REGION Network 6: Mode
   // 0NA,1Manual, 2Auto, 3Step, 4OneCycle, 5Runn, 6Error
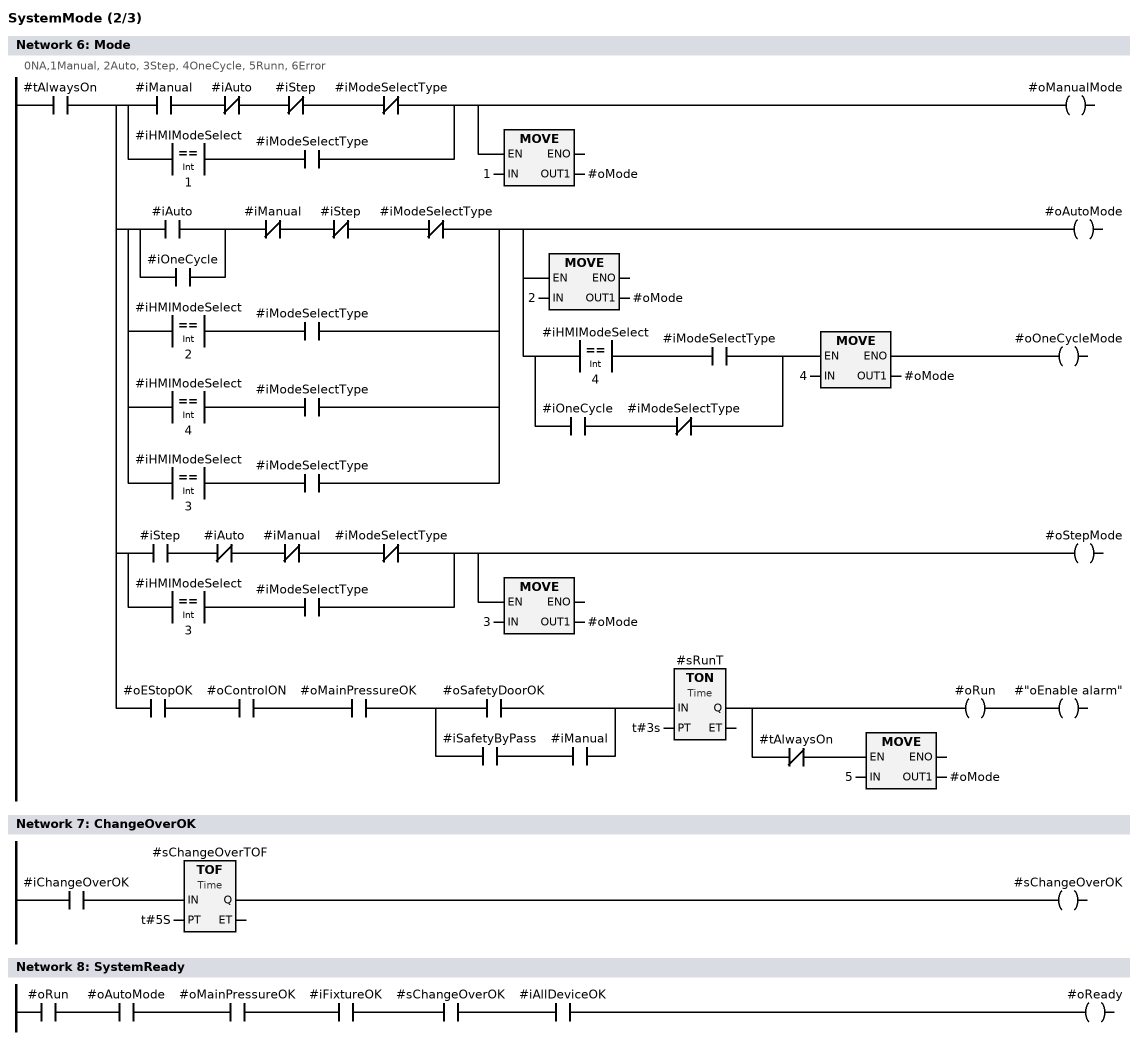
   RUNG wire#powerrail
      Contact( #tAlwaysOn )
      wire#w1
      Contact( #iManual )
      I_Contact( #iAuto )
      I_Contact( #iStep )
      I_Contact( #iModeSelectType )
      wire#w2
      Coil( #oManualMode )
   END_RUNG
   RUNG wire#w1
      { S7_Templates := "SrcType := Int" } EQ_Contact(in1 := #iHMIModeSelect, in2 := 1)
      Contact( #iModeSelectType )
   END_RUNG wire#w2
   RUNG wire#w2
      { S7_GenerateENO := "TRUE" } Move(in := 1, out1 => #oMode)
   END_RUNG
   RUNG wire#w1
      Contact( #iAuto )
      wire#w3
      I_Contact( #iManual )
      I_Contact( #iStep )
      I_Contact( #iModeSelectType )
      wire#w4
      Coil( #oAutoMode )
   END_RUNG
   RUNG wire#w1
      Contact( #iOneCycle )
   END_RUNG wire#w3
   RUNG wire#w1
      { S7_Templates := "SrcType := Int" } EQ_Contact(in1 := #iHMIModeSelect, in2 := 2)
      Contact( #iModeSelectType )
   END_RUNG wire#w4
   RUNG wire#w1
      { S7_Templates := "SrcType := Int" } EQ_Contact(in1 := #iHMIModeSelect, in2 := 4)
      Contact( #iModeSelectType )
   END_RUNG wire#w4
   RUNG wire#w1
      { S7_Templates := "SrcType := Int" } EQ_Contact(in1 := #iHMIModeSelect, in2 := 3)
      Contact( #iModeSelectType )
   END_RUNG wire#w4
   RUNG wire#w4
      { S7_GenerateENO := "TRUE" } Move(in := 2, out1 => #oMode)
   END_RUNG
   RUNG wire#w4
      { S7_Templates := "SrcType := Int" } EQ_Contact(in1 := #iHMIModeSelect, in2 := 4)
      Contact( #iModeSelectType )
      wire#w5
      { S7_GenerateENO := "TRUE" } Move(in := 4, out1 => #oMode)
      Coil( #oOneCycleMode )
   END_RUNG
   RUNG wire#w4
      Contact( #iOneCycle )
      I_Contact( #iModeSelectType )
   END_RUNG wire#w5
   RUNG wire#w1
      Contact( #iStep )
      I_Contact( #iAuto )
      I_Contact( #iManual )
      I_Contact( #iModeSelectType )
      wire#w6
      Coil( #oStepMode )
   END_RUNG
   RUNG wire#w1
      { S7_Templates := "SrcType := Int" } EQ_Contact(in1 := #iHMIModeSelect, in2 := 3)
      Contact( #iModeSelectType )
   END_RUNG wire#w6
   RUNG wire#w6
      { S7_GenerateENO := "TRUE" } Move(in := 3, out1 => #oMode)
   END_RUNG
   RUNG wire#w1
      Contact( #oEStopOK )
      Contact( #oControlON )
      Contact( #oMainPressureOK )
      wire#w7
      Contact( #oSafetyDoorOK )
      wire#w8
      { S7_Templates := "time_type := Time" } #sRunT.TON(pt := t#3s, et =>)
      wire#w9
      Coil( #oRun )
      Coil( #"oEnable alarm" )
   END_RUNG
   RUNG wire#w7
      Contact( #iSafetyByPass )
      Contact( #iManual )
   END_RUNG wire#w8
   RUNG wire#w9
      I_Contact( #tAlwaysOn )
      { S7_GenerateENO := "TRUE" } Move(in := 5, out1 => #oMode)
   END_RUNG
   // the same network as SCL:
   // ENO of a box is taken as its EN; it also drops when the box reports an error
   #oManualMode := #tAlwaysOn AND ((#iManual AND NOT #iAuto AND NOT #iStep AND NOT #iModeSelectType) OR ((#iHMIModeSelect = 1) AND #iModeSelectType));
   IF #oManualMode THEN #oMode := 1; END_IF;
   #oAutoMode := #tAlwaysOn AND (((#iAuto OR #iOneCycle) AND NOT #iManual AND NOT #iStep AND NOT #iModeSelectType) OR ((#iHMIModeSelect = 2) AND #iModeSelectType) OR ((#iHMIModeSelect = 4) AND #iModeSelectType) OR ((#iHMIModeSelect = 3) AND #iModeSelectType));
   IF #oAutoMode THEN #oMode := 2; END_IF;
   #_w1 := #oAutoMode AND (((#iHMIModeSelect = 4) AND #iModeSelectType) OR (#iOneCycle AND NOT #iModeSelectType));
   IF #_w1 THEN #oMode := 4; END_IF;
   #oOneCycleMode := #_w1;
   #oStepMode := #tAlwaysOn AND ((#iStep AND NOT #iAuto AND NOT #iManual AND NOT #iModeSelectType) OR ((#iHMIModeSelect = 3) AND #iModeSelectType));
   IF #oStepMode THEN #oMode := 3; END_IF;
   #sRunT(IN := #tAlwaysOn AND #oEStopOK AND #oControlON AND #oMainPressureOK AND (#oSafetyDoorOK OR (#iSafetyByPass AND #iManual)),   // TON
          PT := t#3s);
   #oRun := #sRunT.Q;
   #"oEnable alarm" := #sRunT.Q;
   IF #sRunT.Q AND NOT #tAlwaysOn THEN #oMode := 5; END_IF;
END_REGION

REGION Network 7: ChangeOverOK
   RUNG wire#powerrail
      Contact( #iChangeOverOK )
      { S7_Templates := "time_type := Time" } #sChangeOverTOF.TOF(pt := t#5S, et =>)
      Coil( #sChangeOverOK )
   END_RUNG
   // the same network as SCL:
   #sChangeOverTOF(IN := #iChangeOverOK, PT := t#5S);   // TOF
   #sChangeOverOK := #sChangeOverTOF.Q;
END_REGION

REGION Network 8: SystemReady
   RUNG wire#powerrail
      Contact( #oRun )
      Contact( #oAutoMode )
      Contact( #oMainPressureOK )
      Contact( #iFixtureOK )
      Contact( #sChangeOverOK )
      Contact( #iAllDeviceOK )
      Coil( #oReady )
   END_RUNG
   // the same network as SCL:
   #oReady := #oRun AND #oAutoMode AND #oMainPressureOK AND #iFixtureOK AND #sChangeOverOK AND #iAllDeviceOK;
END_REGION

REGION Network 9: SystemStatus
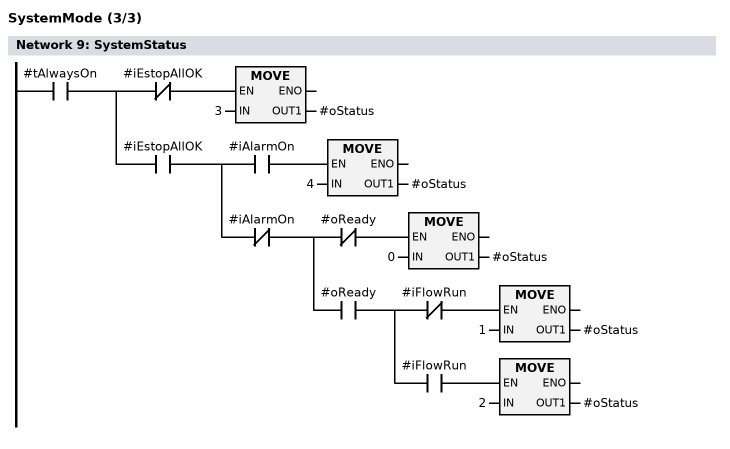
   RUNG wire#powerrail
      Contact( #tAlwaysOn )
      wire#w1
      I_Contact( #iEstopAllOK )
      Move(in := 3, out1 => #oStatus)
   END_RUNG
   RUNG wire#w1
      Contact( #iEstopAllOK )
      wire#w2
      Contact( #iAlarmOn )
      Move(in := 4, out1 => #oStatus)
   END_RUNG
   RUNG wire#w2
      I_Contact( #iAlarmOn )
      wire#w3
      I_Contact( #oReady )
      Move(in := 0, out1 => #oStatus)
   END_RUNG
   RUNG wire#w3
      Contact( #oReady )
      wire#w4
      I_Contact( #iFlowRun )
      Move(in := 1, out1 => #oStatus)
   END_RUNG
   RUNG wire#w4
      Contact( #iFlowRun )
      Move(in := 2, out1 => #oStatus)
   END_RUNG
   // the same network as SCL:
   IF #tAlwaysOn AND NOT #iEstopAllOK THEN #oStatus := 3; END_IF;
   #_w1 := #tAlwaysOn AND #iEstopAllOK;
   IF #_w1 AND #iAlarmOn THEN #oStatus := 4; END_IF;
   #_w2 := #_w1 AND NOT #iAlarmOn;
   IF #_w2 AND NOT #oReady THEN #oStatus := 0; END_IF;
   #_w3 := #_w2 AND #oReady;
   IF #_w3 AND NOT #iFlowRun THEN #oStatus := 1; END_IF;
   IF #_w3 AND #iFlowRun THEN #oStatus := 2; END_IF;
END_REGION
END_FUNCTION_BLOCK

FUNCTION_BLOCK "AutoProcessDataPopUp"   // FB1666, SCL
{ S7_Optimized_Access := 'TRUE' }
// stored: AutoNumber false, MemoryReserve 100, SetENOAutomatically false
   VAR_IN_OUT
      idx { ExternalAccessible := 'False'; ExternalVisible := 'False'; ExternalWritable := 'False'} : Int;
   END_VAR
   VAR_TEMP
      DefaultData : "ProcessData";
   END_VAR
BEGIN
   REGION read me
     // ============================================================================
     // PROGRAM START COMMENT
     // ============================================================================
     // EN:
     // FC_AutoProcessPopup handles popup visualization and editing of AutoProcess
     // data based on index from HMI.
     // The function provides:
     //  - automatic data loading from AutoProcessData according to selected index,
     //  - two-step confirmation for safe data overwrite (compare first, write second),
     //  - automatic reset of edit mode when index is changed,
     //  - delete functionality for selected record,
     //  - status bits for HMI to visualize pending changes and confirmation dialogs,
     //  - index range control (1..16).
     //
     // Data flow:
     // AutoProcessData  -> ActualSHowingData  (display mode)
     // ActualSHowingData -> AutoProcessData  (after double confirmation)
     //
     // Usage:
     // Call cyclically 
     // RMS index is taken from AutoProcess_HMI.IndexProcess.
     //
     // ----------------------------------------------------------------------------
     // CZ:
     // FC_AutoProcessPopup obsluhuje zobrazení a editaci dat AutoProcess podle
     // indexu z HMI.
     // Funkce zajišťuje:
     //  - automatické načítání dat z AutoProcessData podle zvoleného indexu,
     //  - dvoukrokové potvrzení zápisu (nejprve porovnání, poté zápis),
     //  - automatické zrušení editace při změně indexu,
     //  - mazání záznamu podle indexu,
     //  - stavové bity pro HMI (čekající změna, potvrzovací dialog),
     //  - kontrolu rozsahu indexu (1..16).
     //
     // Tok dat:
     // AutoProcessData  -> ActualSHowingData  (zobrazení)
     // ActualSHowingData -> AutoProcessData  (po potvrzení)
     //
     // Použití:
     // Volat cyklicky 
     // Index je čten z AutoProcess_HMI.IndexProcess.
     // ============================================================================

     // Statement section REGION

   END_REGION


   REGION IndexRangeCheck
     // EN: Clamp index to range 1..16
     // CZ: Oříznutí indexu do rozsahu 1..16
     IF #idx < 1 THEN
       #idx := 1;
       "AutoProcess_HMI".IndexProcess := #idx;
     ELSIF #idx > 16 THEN
       #idx := 16;
       "AutoProcess_HMI".IndexProcess := #idx;

     END_IF;
   END_REGION


   REGION IndexHandling
     // ---------------------------------------------------------------------------
     // EN: Detect index change and reset edit session
     // CZ: Detekce změny indexu a zrušení editace
     // ---------------------------------------------------------------------------
     #idx := "AutoProcess_HMI".IndexProcess;

     IF #idx <> "AutoProcess_HMI".Data_handling.LastIndex THEN
       "AutoProcess_HMI".Data_handling.UpdateData_switch := FALSE;
       "AutoProcess_HMI".Data_handling.UpdateData_Confirm := FALSE;
       "AutoProcess_HMI".Data_handling.FinalConfirm_Write := FALSE;
       "AutoProcess_HMI".Data_handling.ConfirmDialogActive := FALSE;
       "AutoProcess_HMI".Data_handling.ChangePending := FALSE;
       "AutoProcess_HMI".Data_handling.DeleteData := FALSE;
       "AutoProcess_HMI".Data_handling.LastIndex := #idx;
     END_IF;
   END_REGION



   REGION ShowData
     // ---------------------------------------------------------------------------
     // EN: Copy data to HMI if edit mode is inactive
     // CZ: Zobrazování dat – pokud není editace, kopíruj data z DB
     // ---------------------------------------------------------------------------
     IF NOT "AutoProcess_HMI".Data_handling.UpdateData_switch THEN
       CASE #idx OF
         1:
           "AutoProcess_HMI".ActualSHowingData := "AutoProcessData".A_ScanRotate;
         2:
           "AutoProcess_HMI".ActualSHowingData := "AutoProcessData".F_Robot1Grip1;
         3:
           "AutoProcess_HMI".ActualSHowingData := "AutoProcessData".F_Robot1Grip2;
         4:
           "AutoProcess_HMI".ActualSHowingData := "AutoProcessData".B_Press1;
         5:
           "AutoProcess_HMI".ActualSHowingData := "AutoProcessData".C_Glue;
         6:
           "AutoProcess_HMI".ActualSHowingData := "AutoProcessData".F_Robot2Grip1;
         7:
           "AutoProcess_HMI".ActualSHowingData := "AutoProcessData".F_Robot2Grip2;
         8:
           "AutoProcess_HMI".ActualSHowingData := "AutoProcessData".C_GlueNGBuffer;
         9:
           "AutoProcess_HMI".ActualSHowingData := "AutoProcessData".C_MagnScanNGBuffer;
         10:
           "AutoProcess_HMI".ActualSHowingData := "AutoProcessData".B_Press2;
         11:
           "AutoProcess_HMI".ActualSHowingData := "AutoProcessData".F_Robot3Grip1;
         12:
           "AutoProcess_HMI".ActualSHowingData := "AutoProcessData".F_Robot3Grip2;
         13:
           "AutoProcess_HMI".ActualSHowingData := "AutoProcessData".H_ShafeLine;
         14:
           "AutoProcess_HMI".ActualSHowingData := "AutoProcessData".J_ShafeLine;
         15:
           "AutoProcess_HMI".ActualSHowingData := "AutoProcessData".K_ShafeLine;
         16:
           "AutoProcess_HMI".ActualSHowingData := "AutoProcessData".L_ShafeLine;
         ELSE
           ;
           // EN: invalid index / CZ: neplatný index
       END_CASE;
     END_IF;
   END_REGION



   REGION FirstConfirm
     // ---------------------------------------------------------------------------
     // EN: First confirmation → enable compare dialog
     // CZ: První potvrzení → aktivace porovnávacího dialogu
     // ---------------------------------------------------------------------------
     IF "AutoProcess_HMI".Data_handling.UpdateData_switch
       AND "AutoProcess_HMI".Data_handling.UpdateData_Confirm
       AND NOT "AutoProcess_HMI".Data_handling.ConfirmDialogActive THEN

       "AutoProcess_HMI".Data_handling.ConfirmDialogActive := TRUE;
       "AutoProcess_HMI".Data_handling.ChangePending := TRUE;

       "AutoProcess_HMI".Data_handling.UpdateData_Confirm := FALSE;
     END_IF;
   END_REGION



   REGION FinalWrite
     // ---------------------------------------------------------------------------
     // EN: Final confirmation → write to data DB
     // CZ: Finální potvrzení → zápis do DB
     // ---------------------------------------------------------------------------
     IF "AutoProcess_HMI".Data_handling.ConfirmDialogActive
       AND "AutoProcess_HMI".Data_handling.FinalConfirm_Write THEN

       CASE #idx OF
         1:
           "AutoProcessData".A_ScanRotate := "AutoProcess_HMI".ActualSHowingData;
         2:
           "AutoProcessData".F_Robot1Grip1 := "AutoProcess_HMI".ActualSHowingData;
         3:
           "AutoProcessData".F_Robot1Grip2 := "AutoProcess_HMI".ActualSHowingData;
         4:
           "AutoProcessData".B_Press1 := "AutoProcess_HMI".ActualSHowingData;
         5:
           "AutoProcessData".C_Glue := "AutoProcess_HMI".ActualSHowingData;
         6:
           "AutoProcessData".F_Robot2Grip1 := "AutoProcess_HMI".ActualSHowingData;
         7:
           "AutoProcessData".F_Robot2Grip2 := "AutoProcess_HMI".ActualSHowingData;
         8:
           "AutoProcessData".C_GlueNGBuffer := "AutoProcess_HMI".ActualSHowingData;
         9:
           "AutoProcessData".C_MagnScanNGBuffer := "AutoProcess_HMI".ActualSHowingData;
         10:
           "AutoProcessData".B_Press2 := "AutoProcess_HMI".ActualSHowingData;
         11:
           "AutoProcessData".F_Robot3Grip1 := "AutoProcess_HMI".ActualSHowingData;
         12:
           "AutoProcessData".F_Robot3Grip2 := "AutoProcess_HMI".ActualSHowingData;
         13:
           "AutoProcessData".H_ShafeLine := "AutoProcess_HMI".ActualSHowingData;
         14:
           "AutoProcessData".J_ShafeLine := "AutoProcess_HMI".ActualSHowingData;
         15:
           "AutoProcessData".K_ShafeLine := "AutoProcess_HMI".ActualSHowingData;
         16:
           "AutoProcessData".L_ShafeLine := "AutoProcess_HMI".ActualSHowingData;
         ELSE
           ;
       END_CASE;

       // reset flags after write
       "AutoProcess_HMI".Data_handling.ConfirmDialogActive := FALSE;
       "AutoProcess_HMI".Data_handling.ChangePending := FALSE;
       "AutoProcess_HMI".Data_handling.FinalConfirm_Write := FALSE;
       "AutoProcess_HMI".Data_handling.UpdateData_switch := FALSE;
     END_IF;
   END_REGION



   REGION DeleteData
     // ---------------------------------------------------------------------------
     // EN: Delete selected Record (reset to default struct)
     // CZ: Smazání záznamu – vynulování struktury
     // ---------------------------------------------------------------------------
     IF "AutoProcess_HMI".Data_handling.DeleteData AND
       "AutoProcess_HMI".Data_handling.FinalConfirm_Write
       THEN

       CASE #idx OF
         1:
           "AutoProcessData".A_ScanRotate := #DefaultData;
         2:
           "AutoProcessData".F_Robot1Grip1 := #DefaultData;
         3:
           "AutoProcessData".F_Robot1Grip2 := #DefaultData;
         4:
           "AutoProcessData".B_Press1 := #DefaultData;
         5:
           "AutoProcessData".C_Glue := #DefaultData;
         6:
           "AutoProcessData".F_Robot2Grip1 := #DefaultData;
         7:
           "AutoProcessData".F_Robot2Grip2 := #DefaultData;
         8:
           "AutoProcessData".C_GlueNGBuffer := #DefaultData;
         9:
           "AutoProcessData".C_MagnScanNGBuffer := #DefaultData;
         10:
           "AutoProcessData".B_Press2 := #DefaultData;
         11:
           "AutoProcessData".F_Robot3Grip1 := #DefaultData;
         12:
           "AutoProcessData".F_Robot3Grip2 := #DefaultData;
         13:
           "AutoProcessData".H_ShafeLine := #DefaultData;
         14:
           "AutoProcessData".J_ShafeLine := #DefaultData;
         15:
           "AutoProcessData".K_ShafeLine := #DefaultData;
         16:
           "AutoProcessData".L_ShafeLine := #DefaultData;
         ELSE
           ;
       END_CASE;

       // reset delete + editing states
       "AutoProcess_HMI".Data_handling.DeleteData := FALSE;
       "AutoProcess_HMI".Data_handling.UpdateData_switch := FALSE;
       "AutoProcess_HMI".Data_handling.UpdateData_Confirm := FALSE;
       "AutoProcess_HMI".Data_handling.FinalConfirm_Write := FALSE;
       "AutoProcess_HMI".Data_handling.ConfirmDialogActive := FALSE;
       "AutoProcess_HMI".Data_handling.ChangePending := FALSE;
     END_IF;
   END_REGION

   REGION StationProductIcons
     // EN: Set icon bits if station contains product (PartStatus <> 0)
     // CZ: Nastavení bitů ikony – stanice má kus, pokud PartStatus <> 0

     // 1 – A_ScanRotate
     "AutoProcess_HMI".StationHasProduct[1] :=
     "AutoProcessData".A_ScanRotate.PartStatus <> 0;

     // 2 – F_Robot1Grip1
     "AutoProcess_HMI".StationHasProduct[2] :=
     "AutoProcessData".F_Robot1Grip1.PartStatus <> 0;

     // 3 – F_Robot1Grip2
     "AutoProcess_HMI".StationHasProduct[3] :=
     "AutoProcessData".F_Robot1Grip2.PartStatus <> 0;

     // 4 – B_Press1
     "AutoProcess_HMI".StationHasProduct[4] :=
     "AutoProcessData".B_Press1.PartStatus <> 0;

     // 5 – C_Glue
     "AutoProcess_HMI".StationHasProduct[5] :=
     "AutoProcessData".C_Glue.PartStatus <> 0;

     // 6 – F_Robot2Grip1
     "AutoProcess_HMI".StationHasProduct[6] :=
     "AutoProcessData".F_Robot2Grip1.PartStatus <> 0;

     // 7 – F_Robot2Grip2
     "AutoProcess_HMI".StationHasProduct[7] :=
     "AutoProcessData".F_Robot2Grip2.PartStatus <> 0;

     // 8 – C_GlueNGBuffer
     "AutoProcess_HMI".StationHasProduct[8] :=
     "AutoProcessData".C_GlueNGBuffer.PartStatus <> 0;

     // 9 – C_MagnScanNGBuffer
     "AutoProcess_HMI".StationHasProduct[9] :=
     "AutoProcessData".C_MagnScanNGBuffer.PartStatus <> 0;

     // 10 – B_Press2
     "AutoProcess_HMI".StationHasProduct[10] :=
     "AutoProcessData".B_Press2.PartStatus <> 0;

     // 11 – F_Robot3Grip1
     "AutoProcess_HMI".StationHasProduct[11] :=
     "AutoProcessData".F_Robot3Grip1.PartStatus <> 0;

     // 12 – F_Robot3Grip2
     "AutoProcess_HMI".StationHasProduct[12] :=
     "AutoProcessData".F_Robot3Grip2.PartStatus <> 0;

     // 13 – H_ShafeLine
     "AutoProcess_HMI".StationHasProduct[13] :=
     "AutoProcessData".H_ShafeLine.PartStatus <> 0;

     // 14 – J_ShafeLine
     "AutoProcess_HMI".StationHasProduct[14] :=
     "AutoProcessData".J_ShafeLine.PartStatus <> 0;

     // 15 – K_ShafeLine
     "AutoProcess_HMI".StationHasProduct[15] :=
     "AutoProcessData".K_ShafeLine.PartStatus <> 0;

     // 16 – L_ShafeLine
     "AutoProcess_HMI".StationHasProduct[16] :=
     "AutoProcessData".L_ShafeLine.PartStatus <> 0;

   END_REGION
END_FUNCTION_BLOCK

ORGANIZATION_BLOCK "02_Warm Restart"   // OB100, LAD, Startup
TITLE = "Complete Restart"
{ S7_Optimized_Access := 'FALSE' }
AUTHOR : RCS
// 1.该部分用户可以根据系统的需要将CPU第一次扫描需要执行的逻辑写在此处
// stored: AutoNumber false, SetENOAutomatically false
   VAR_TEMP
      OB100_EV_CLASS : Byte;   // 16#13, Event class 1, Entering event state, Event logged in diagnostic buffer
      OB100_STRTUP : Byte;   // 16#81/82/83/84 Method of startup
      OB100_PRIORITY : Byte;   // Priority of OB Execution
      OB100_OB_NUMBR : Byte;   // 100 (Organization block 100, OB100)
      OB100_RESERVED_1 : Byte;   // Reserved for system
      OB100_RESERVED_2 : Byte;   // Reserved for system
      OB100_STOP : Word;   // Event that caused CPU to stop (16#4xxx)
      OB100_STRT_INFO : DWord;   // Information on how system started
      OB100_DATE_TIME : Date_And_Time;   // Date and time OB100 started
   END_VAR
BEGIN

REGION Network 1
   // 系统程序段无需改动
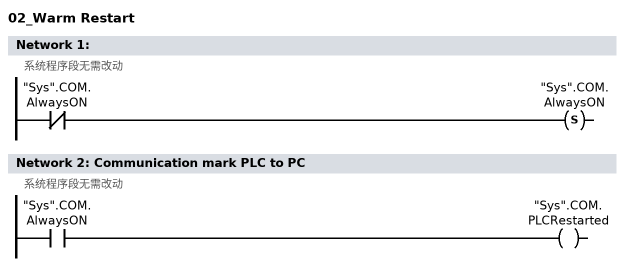
   RUNG wire#powerrail
      I_Contact( "Sys".COM.AlwaysON )
      S_Coil( "Sys".COM.AlwaysON )
   END_RUNG
   // the same network as SCL:
   IF NOT "Sys".COM.AlwaysON THEN "Sys".COM.AlwaysON := TRUE; END_IF;
END_REGION

REGION Network 2: Communication mark PLC to PC
   // 系统程序段无需改动
   RUNG wire#powerrail
      Contact( "Sys".COM.AlwaysON )
      Coil( "Sys".COM.PLCRestarted )
   END_RUNG
   // the same network as SCL:
   "Sys".COM.PLCRestarted := "Sys".COM.AlwaysON;
END_REGION

NETWORK
TITLE = 

      L     1;
      T     "Station_Sys".Status.ModeSV;

END_ORGANIZATION_BLOCK

ORGANIZATION_BLOCK "03_CYC_INT2"   // OB32, LAD, CyclicInterrupt
TITLE = "Cyclic Interrupt"
{ S7_Optimized_Access := 'FALSE' }
// stored: AutoNumber false, SetENOAutomatically false
   VAR_TEMP
      OB32_EV_CLASS : Byte;   // Bits 0-3 = 1 (Coming event), Bits 4-7 = 1 (Event class 1)
      OB32_STRT_INF : Byte;   // 16#33 (OB 32 has started)
      OB32_PRIORITY : Byte;   // Priority of OB Execution
      OB32_OB_NUMBR : Byte;   // 32 (Organization block 32, OB32)
      OB32_RESERVED_1 : Byte;   // Reserved for system
      OB32_RESERVED_2 : Byte;   // Reserved for system
      OB32_PHS_OFFSET : Int;   // Phase offset (integer, milliseconds)
      OB32_RESERVED_3 : Int;   // Reserved for system
      OB32_EXC_FREQ : Int;   // Frequency of execution (msec)
      OB32_DATE_TIME : Date_And_Time;   // Date and time OB32 started
   END_VAR
BEGIN

REGION Network 1
   // //Keep resource code
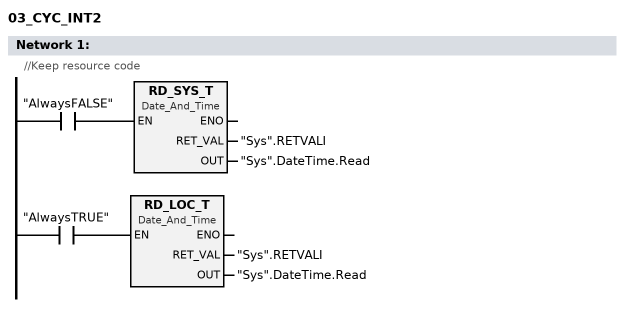
   RUNG wire#powerrail
      Contact( "AlwaysFALSE" )
      { S7_Templates := "date_type := Date_And_Time" } RD_SYS_T(RET_VAL => "Sys".RETVALI, OUT => "Sys".DateTime.Read)
   END_RUNG
   RUNG wire#powerrail
      Contact( "AlwaysTRUE" )
      { S7_Templates := "date_type := Date_And_Time" } RD_LOC_T(RET_VAL => "Sys".RETVALI, OUT => "Sys".DateTime.Read)
   END_RUNG
   // the same network as SCL:
   IF "AlwaysFALSE" THEN "Sys".RETVALI := RD_SYS_T(OUT => "Sys".DateTime.Read); END_IF;
   IF "AlwaysTRUE" THEN "Sys".RETVALI := RD_LOC_T(OUT => "Sys".DateTime.Read); END_IF;
END_REGION

NETWORK
TITLE = Diagnostic
//      CALL  "Diagnostic"
//         iCPUType :=2
//         iDBNum   :=3001
//         iOffset  :=0


END_ORGANIZATION_BLOCK

ORGANIZATION_BLOCK "04_CYC_INT5"   // OB35, LAD, CyclicInterrupt
TITLE = "Cyclic Interrupt"
{ S7_Optimized_Access := 'FALSE' }
// stored: AutoNumber false, SetENOAutomatically false
   VAR_TEMP
      OB35_EV_CLASS : Byte;   // Bits 0-3 = 1 (Coming event), Bits 4-7 = 1 (Event class 1)
      OB35_STRT_INF : Byte;   // 16#36 (OB 35 has started)
      OB35_PRIORITY : Byte;   // Priority of OB Execution
      OB35_OB_NUMBR : Byte;   // 35 (Organization block 35, OB35)
      OB35_RESERVED_1 : Byte;   // Reserved for system
      OB35_RESERVED_2 : Byte;   // Reserved for system
      OB35_PHASE_OFFSET : Word;   // Phase offset (msec)
      OB35_RESERVED_3 : Int;   // Reserved for system
      OB35_EXC_FREQ : Int;   // Frequency of execution (msec)
      OB35_DATE_TIME : Date_And_Time;   // Date and time OB35 started
   END_VAR
BEGIN
END_ORGANIZATION_BLOCK

ORGANIZATION_BLOCK "05_MOD_ERR"   // OB122, STL, IOAccessError
TITLE = "Module Access Error"
{ S7_Optimized_Access := 'FALSE' }
   VAR_TEMP
      OB122_EV_CLASS : Byte;   // 16#29, Event class 2, Entering event state, Internal fault event
      OB122_SW_FLT : Byte;   // 16#XX Software error code
      OB122_PRIORITY : Byte;   // Priority of OB Execution
      OB122_OB_NUMBR : Byte;   // 122 (Organization block 122, OB122)
      OB122_BLK_TYPE : Byte;   // 16#88/8C/8E Type of block fault occured in
      OB122_MEM_AREA : Byte;   // Memory area where access error occured
      OB122_MEM_ADDR : Word;   // Memory address where access error occured
      OB122_BLK_NUM : Word;   // Block number in which error occured
      OB122_PRG_ADDR : Word;   // Program address where error occured
      OB122_DATE_TIME : Date_And_Time;   // Date and time OB1 started
   END_VAR
BEGIN
END_ORGANIZATION_BLOCK

ORGANIZATION_BLOCK "07_CYCL_FLT"   // OB80, STL, TimeErrorInterrupt
TITLE = "Cycle Time Fault"
{ S7_Optimized_Access := 'FALSE' }
   VAR_TEMP
      OB80_EV_CLASS : Byte;   // 16#35, Event class 3, Entering event state, Internal fault event
      OB80_FLT_ID : Byte;   // 16#XX, Fault identifcation code
      OB80_PRIORITY : Byte;   // Priority of OB Execution
      OB80_OB_NUMBR : Byte;   // 80 (Organization block 80, OB80)
      OB80_RESERVED_1 : Byte;   // Reserved for system
      OB80_RESERVED_2 : Byte;   // Reserved for system
      OB80_ERROR_INFO : Word;   // Error information on event
      OB80_ERR_EV_CLASS : Byte;   // Class of event causing error
      OB80_ERR_EV_NUM : Byte;   // Number of event causing error
      OB80_OB_PRIORITY : Byte;   // Priority of OB causing error
      OB80_OB_NUM : Byte;   // Number of OB causing error
      OB80_DATE_TIME : Date_And_Time;   // Date and time OB80 started
   END_VAR
BEGIN
END_ORGANIZATION_BLOCK

ORGANIZATION_BLOCK "08_HW_INT0"   // OB40, LAD, HardwareInterrupt
TITLE = "Hardware Interrupt"
{ S7_Optimized_Access := 'FALSE' }
// stored: AutoNumber false, SetENOAutomatically false
   VAR_TEMP
      OB40_EV_CLASS : Byte;   // Bits 0-3 = 1 (Coming event), Bits 4-7 = 1 (Event class 1)
      OB40_STRT_INF : Byte;   // 16#41 (OB 40 has started)
      OB40_PRIORITY : Byte;   // Priority of OB Execution
      OB40_OB_NUMBR : Byte;   // 40 (Organization block 40, OB40)
      OB40_RESERVED_1 : Byte;   // Reserved for system
      OB40_IO_FLAG : Byte;   // 16#54 (input module), 16#55 (output module)
      OB40_MDL_ADDR : Word;   // Base address of module initiating interrupt
      OB40_POINT_ADDR : DWord;   // Interrupt status of the module
      OB40_DATE_TIME : Date_And_Time;   // Date and time OB40 started
   END_VAR
BEGIN
END_ORGANIZATION_BLOCK

ORGANIZATION_BLOCK "09_I/O_FLT1"   // OB82, STL, DiagnosticErrorInterrupt
TITLE = "I/O Point Fault"
{ S7_Optimized_Access := 'FALSE' }
   VAR_TEMP
      OB82_EV_CLASS : Byte;   // 16#39, Event class 3, Entering event state, Internal fault event
      OB82_FLT_ID : Byte;   // 16#XX, Fault identifcation code
      OB82_PRIORITY : Byte;   // Priority of OB Execution
      OB82_OB_NUMBR : Byte;   // 82 (Organization block 82, OB82)
      OB82_RESERVED_1 : Byte;   // Reserved for system
      OB82_IO_FLAG : Byte;   // Input (01010100), Output (01010101)
      OB82_MDL_ADDR : Int;   // Base address of module with fault
      OB82_MDL_DEFECT : Bool;   // Module defective
      OB82_INT_FAULT : Bool;   // Internal fault
      OB82_EXT_FAULT : Bool;   // External fault
      OB82_PNT_INFO : Bool;   // Point information
      OB82_EXT_VOLTAGE : Bool;   // External voltage low
      OB82_FLD_CONNCTR : Bool;   // Field wiring connector missing
      OB82_NO_CONFIG : Bool;   // Module has no configuration data
      OB82_CONFIG_ERR : Bool;   // Module has configuration error
      OB82_MDL_TYPE : Byte;   // Type of module
      OB82_SUB_NDL_ERR : Bool;   // Sub-Module is missing or has error
      OB82_COMM_FAULT : Bool;   // Communication fault
      OB82_MDL_STOP : Bool;   // Module is stopped
      OB82_WTCH_DOG_FLT : Bool;   // Watch dog timer stopped module
      OB82_INT_PS_FLT : Bool;   // Internal power supply fault
      OB82_PRIM_BATT_FLT : Bool;   // Primary battery is in fault
      OB82_BCKUP_BATT_FLT : Bool;   // Backup battery is in fault
      OB82_RESERVED_2 : Bool;   // Reserved for system
      OB82_RACK_FLT : Bool;   // Rack fault, only for bus interface module
      OB82_PROC_FLT : Bool;   // Processor fault
      OB82_EPROM_FLT : Bool;   // EPROM fault
      OB82_RAM_FLT : Bool;   // RAM fault
      OB82_ADU_FLT : Bool;   // ADU fault
      OB82_FUSE_FLT : Bool;   // Fuse fault
      OB82_HW_INTR_FLT : Bool;   // Hardware interupt input in fault
      OB82_RESERVED_3 : Bool;   // Reserved for system
      OB82_DATE_TIME : Date_And_Time;   // Date and time OB82 started
   END_VAR
BEGIN
END_ORGANIZATION_BLOCK

ORGANIZATION_BLOCK "11_PROG_ERR"   // OB121, STL, ProgrammingError
TITLE = "Programming Error"
{ S7_Optimized_Access := 'FALSE' }
   VAR_TEMP
      OB121_EV_CLASS : Byte;   // 16#25, Event class 2, Entering event state, Internal fault event
      OB121_SW_FLT : Byte;   // 16#XX Software programming fault
      OB121_PRIORITY : Byte;   // Priority of OB Execution
      OB121_OB_NUMBR : Byte;   // 121 (Organization block 121, OB121)
      OB121_BLK_TYPE : Byte;   // 16#88/8A/8B/8C/8E Type of block fault occured in
      OB121_RESERVED_1 : Byte;   // Reserved for system
      OB121_FLT_REG : Word;   // 16#XX Specific register that caused fault
      OB121_BLK_NUM : Word;   // Number of block that programming fault occured in
      OB121_PRG_ADDR : Word;   // Address in block where programming fault occured
      OB121_DATE_TIME : Date_And_Time;   // Date and time OB121 started
   END_VAR
BEGIN
END_ORGANIZATION_BLOCK

ORGANIZATION_BLOCK "12_RACK_FLT"   // OB86, STL, RackOrStationFailure
TITLE = "Loss Of Rack Fault"
{ S7_Optimized_Access := 'FALSE' }
   VAR_TEMP
      OB86_EV_CLASS : Byte;   // 16#38/39 Event class 3
      OB86_FLT_ID : Byte;   // 16#C1/C4/C5, Fault identifcation code
      OB86_PRIORITY : Byte;   // Priority of OB Execution
      OB86_OB_NUMBR : Byte;   // 86 (Organization block 86, OB86)
      OB86_RESERVED_1 : Byte;   // Reserved for system
      OB86_RESERVED_2 : Byte;   // Reserved for system
      OB86_MDL_ADDR : Word;   // Base address of IM module in rack with fault
      OB86_RACKS_FLTD : Array[0..31] of Bool;
      OB86_DATE_TIME : Date_And_Time;   // Date and time OB86 started
   END_VAR
BEGIN
END_ORGANIZATION_BLOCK

FUNCTION "fcFixtureCheck" : Void   // FC2, LAD
{ S7_Optimized_Access := 'TRUE' }
// stored: SetENOAutomatically false
   VAR_INPUT
      iRecipeSetValue : Byte;   // 配方设定工装值
   END_VAR
   VAR_IN_OUT
      FixtureIDCheck : Struct
         FixtureIDSetValue : Int;
         FixtureIDCheckValue : Int;
         FixtureCheckResult : Bool;
         FixtureCheckUnEnable : Bool;   // 工装检测使能,不需要检测时，给1
      END_STRUCT;
   END_VAR
BEGIN

REGION Network 2: 配方设定工装值 / Formula set tooling values
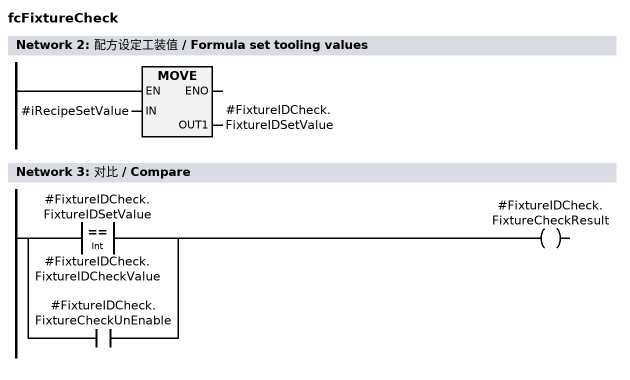
   RUNG wire#powerrail
      Move(in := #iRecipeSetValue, out1 => #FixtureIDCheck.FixtureIDSetValue)
   END_RUNG
   // the same network as SCL:
   #FixtureIDCheck.FixtureIDSetValue := #iRecipeSetValue;
END_REGION

REGION Network 3: 对比 / Compare
   RUNG wire#powerrail
      { S7_Templates := "SrcType := Int" } EQ_Contact(in1 := #FixtureIDCheck.FixtureIDSetValue, in2 := #FixtureIDCheck.FixtureIDCheckValue)
      wire#w1
      Coil( #FixtureIDCheck.FixtureCheckResult )
   END_RUNG
   RUNG wire#powerrail
      Contact( #FixtureIDCheck.FixtureCheckUnEnable )
   END_RUNG wire#w1
   // the same network as SCL:
   #FixtureIDCheck.FixtureCheckResult := (#FixtureIDCheck.FixtureIDSetValue = #FixtureIDCheck.FixtureIDCheckValue) OR #FixtureIDCheck.FixtureCheckUnEnable;
END_REGION
END_FUNCTION

FUNCTION "CylinderModule_V2" : Void   // FC3010, LAD
TITLE = Title
{ S7_Optimized_Access := 'FALSE' }
VERSION : 2.0
// //---------------------------------------------------------------//
// //FunctionName:CylinderV2
// //FunctionDescription:CylinderControl
// //---------------------------------------------------------------//
// //in:
// 
// 	iReset	Bool			reset action
// 	iRun	Bool			system run
// 	iE_stop	Bool			e_stop monitor
// 	iManualMode	Bool		manual mode
// 	iAutoMode	Bool		auto mode
// 	iEnableAlarm	Bool		alarm will popup up
// 	iPulse_100mS	Bool		pulse *100ms
// 	iPulse_1S	Bool		pulse*1s
// 	iCyDBNO	Int	Int		Interface data block number
// 	iCyCounts	Int		total counts of cylinder to be used[must                                                                                                             be>=1 and <=100]
// 
// //inout:
// //out:
// //---------------------------------------------------------------//
// //Version:V2
// //D&T:2016-11-14
// //Group:RCS
// //Author:JM
// //-------------------------Modify1----------------------------------//
// //Version:
// //D&T:2016-11-17
// //Group: RCS
// //Author:
// //Modify:Update cylinder no as output interface
// //-------------------------Modify2----------------------------------//
// //Version:
// //D&T:2022-12-07
// //Group: RCS
// //Author:JM
// //Modify: add action time
// stored: AutoNumber false, SetENOAutomatically false
   VAR_INPUT
      iReset : Bool;   // reset action
      iRun : Bool;   // system run
      iEStop : Bool;   // e_stop monitor
      iManualMode : Bool;   // manual mode
      iAutoMode : Bool;   // auto mode
      iEnableAlarm : Bool;   // alarm will popup up
      iPulse100mS : Bool;   // pulse *100ms
      iPulse1S : Bool;   // pulse*1s
      iError : Bool;   // Outer error force output off
      iGoWorkInterlock : Bool;   // 1=permit motion
      iGoHomeInterlock : Bool;   // 1=permit motion
      iWorkPositionSensor : Bool;   // PLC DI
      iHomePositionSensor : Bool;   // PLC DI
      iValveType : Bool;   // reserve 2022-12-07 / 0 : don`t need holding(2way&3way middle sealing) / 1: need holding(3way middle leaking)
      iManualOutputType : Bool;   // 0 : Output not hold / 1: Output hold (in Manual mode)
      iFaultTime : Int;   // Value*100mS
      iOnPositionTime : Int;   // Value*100mS
   END_VAR
   VAR_OUTPUT
      oGoWP_ButtonActive : Bool;   // For HMI button,indicate can operate go work button
      oGoHP_ButtonActive : Bool;   // For HMI button,indicate can operate go home button
      oCyNo : Byte;
   END_VAR
   VAR_IN_OUT
      ioManualGoWork : Bool;
      ioManualGoHome : Bool;
      ioAutoGoWork : Bool;
      ioAutoGoHome : Bool;
      ioResetOut : Bool;
      ioGoWorkTime : Int;   // Time for going to work position
      ioGoHomeTime : Int;   // time for going to home position
      ioWorkFaultTime : Int;
      ioHomeFaultTime : Int;
      ioBothSensorOnTime : Int;
      ioPulse100mSP : Bool;
      ioAutoGoWorkP : Bool;
      ioAutoGoHomeP : Bool;
      ioGoWork100mSP : Bool;
      ioGoHome100mSP : Bool;
      ioBothSensorOn100mSP : Bool;
      ioAlarm : Bool;
      ioSpare1 : Bool;
      ioSpare2 : Byte;
      ioGoWorkFault : Bool;
      ioGoHomeFault : Bool;
      ioSensorPositionFault : Bool;
      ioGoWorkPosition : Bool;   // PLC DQ
      ioGoHomePosition : Bool;   // PLC DQ
   END_VAR
   VAR_TEMP   // added for the SCL form of the ladder/FBD networks
      _w1 : Bool;
      _w2 : Bool;
      _w3 : Bool;
      _w4 : Bool;
   END_VAR
BEGIN

REGION Network 1: Reset Go Work & Go Home
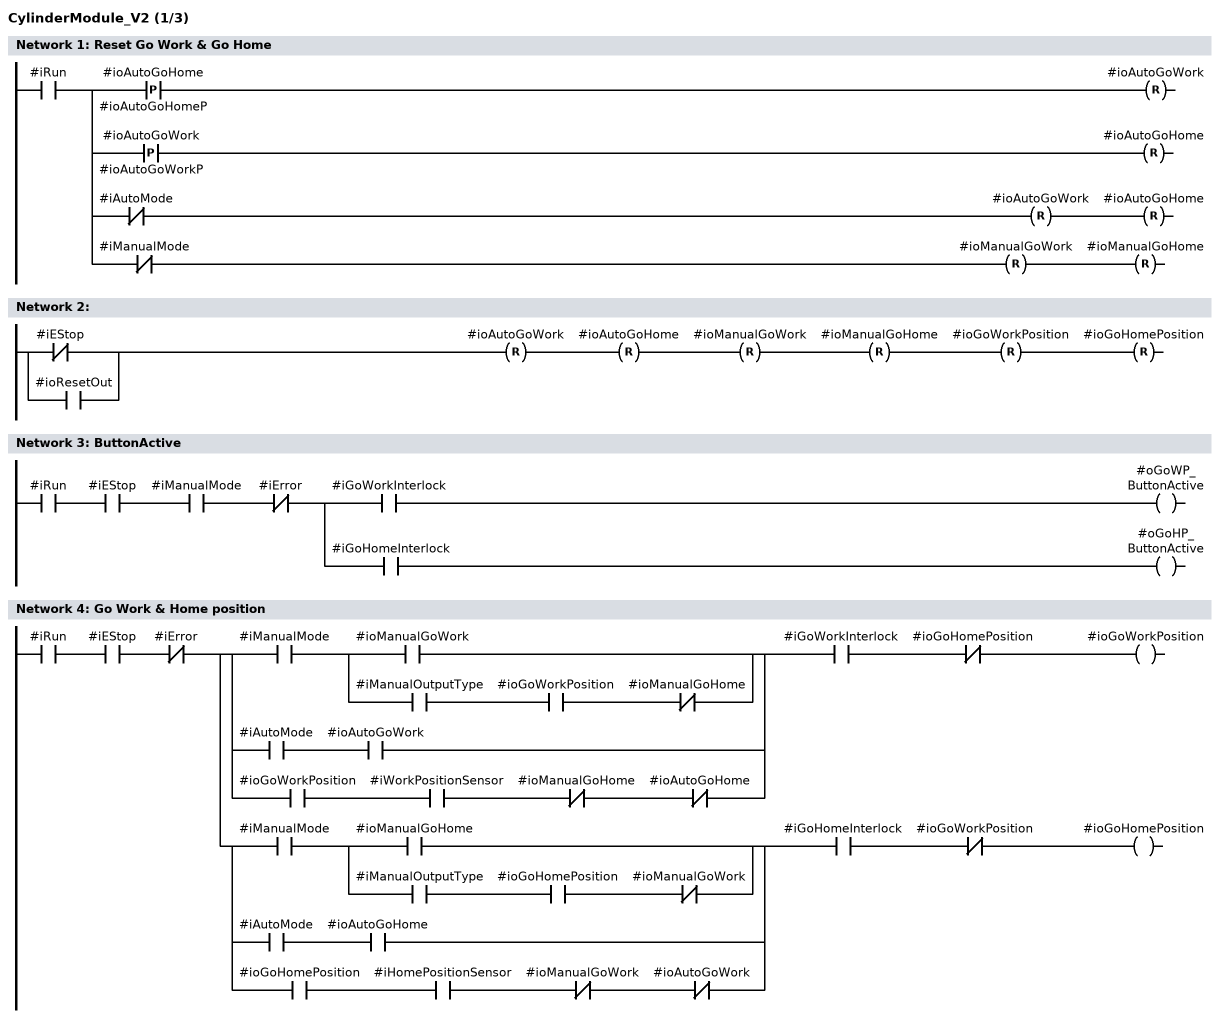
   RUNG wire#powerrail
      Contact( #iRun )
      wire#w1
      P_Contact(operand := #ioAutoGoHome, bit := #ioAutoGoHomeP)
      R_Coil( #ioAutoGoWork )
   END_RUNG
   RUNG wire#w1
      P_Contact(operand := #ioAutoGoWork, bit := #ioAutoGoWorkP)
      R_Coil( #ioAutoGoHome )
   END_RUNG
   RUNG wire#w1
      I_Contact( #iAutoMode )
      R_Coil( #ioAutoGoWork )
      R_Coil( #ioAutoGoHome )
   END_RUNG
   RUNG wire#w1
      I_Contact( #iManualMode )
      R_Coil( #ioManualGoWork )
      R_Coil( #ioManualGoHome )
   END_RUNG
   // the same network as SCL:
   #_w1 := #iRun AND #ioAutoGoHome AND NOT #ioAutoGoHomeP;   // rising edge of #ioAutoGoHome
   #ioAutoGoHomeP := #ioAutoGoHome;
   IF #_w1 THEN #ioAutoGoWork := FALSE; END_IF;
   #_w2 := #iRun AND #ioAutoGoWork AND NOT #ioAutoGoWorkP;   // rising edge of #ioAutoGoWork
   #ioAutoGoWorkP := #ioAutoGoWork;
   IF #_w2 THEN #ioAutoGoHome := FALSE; END_IF;
   IF #iRun AND NOT #iAutoMode THEN
       #ioAutoGoWork := FALSE;
       #ioAutoGoHome := FALSE;
   END_IF;
   IF #iRun AND NOT #iManualMode THEN
       #ioManualGoWork := FALSE;
       #ioManualGoHome := FALSE;
   END_IF;
END_REGION

REGION Network 2
   RUNG wire#powerrail
      I_Contact( #iEStop )
      wire#w1
      R_Coil( #ioAutoGoWork )
      R_Coil( #ioAutoGoHome )
      R_Coil( #ioManualGoWork )
      R_Coil( #ioManualGoHome )
      R_Coil( #ioGoWorkPosition )
      R_Coil( #ioGoHomePosition )
   END_RUNG
   RUNG wire#powerrail
      Contact( #ioResetOut )
   END_RUNG wire#w1
   // the same network as SCL:
   IF NOT #iEStop OR #ioResetOut THEN
       #ioAutoGoWork := FALSE;
       #ioAutoGoHome := FALSE;
       #ioManualGoWork := FALSE;
       #ioManualGoHome := FALSE;
       #ioGoWorkPosition := FALSE;
       #ioGoHomePosition := FALSE;
   END_IF;
END_REGION

REGION Network 3: ButtonActive
   RUNG wire#powerrail
      Contact( #iRun )
      Contact( #iEStop )
      Contact( #iManualMode )
      I_Contact( #iError )
      wire#w1
      Contact( #iGoWorkInterlock )
      Coil( #oGoWP_ButtonActive )
   END_RUNG
   RUNG wire#w1
      Contact( #iGoHomeInterlock )
      Coil( #oGoHP_ButtonActive )
   END_RUNG
   // the same network as SCL:
   #_w1 := #iRun AND #iEStop AND #iManualMode AND NOT #iError;
   #oGoWP_ButtonActive := #_w1 AND #iGoWorkInterlock;
   #oGoHP_ButtonActive := #_w1 AND #iGoHomeInterlock;
END_REGION

REGION Network 4: Go Work & Home position
   RUNG wire#powerrail
      Contact( #iRun )
      Contact( #iEStop )
      I_Contact( #iError )
      wire#w1
      Contact( #iManualMode )
      wire#w2
      Contact( #ioManualGoWork )
      wire#w3
      Contact( #iGoWorkInterlock )
      I_Contact( #ioGoHomePosition )
      Coil( #ioGoWorkPosition )
   END_RUNG
   RUNG wire#w2
      Contact( #iManualOutputType )
      Contact( #ioGoWorkPosition )
      I_Contact( #ioManualGoHome )
   END_RUNG wire#w3
   RUNG wire#w1
      Contact( #iAutoMode )
      Contact( #ioAutoGoWork )
   END_RUNG wire#w3
   RUNG wire#w1
      Contact( #ioGoWorkPosition )
      Contact( #iWorkPositionSensor )
      I_Contact( #ioManualGoHome )
      I_Contact( #ioAutoGoHome )
   END_RUNG wire#w3
   RUNG wire#w1
      Contact( #iManualMode )
      wire#w4
      Contact( #ioManualGoHome )
      wire#w5
      Contact( #iGoHomeInterlock )
      I_Contact( #ioGoWorkPosition )
      Coil( #ioGoHomePosition )
   END_RUNG
   RUNG wire#w4
      Contact( #iManualOutputType )
      Contact( #ioGoHomePosition )
      I_Contact( #ioManualGoWork )
   END_RUNG wire#w5
   RUNG wire#w1
      Contact( #iAutoMode )
      Contact( #ioAutoGoHome )
   END_RUNG wire#w5
   RUNG wire#w1
      Contact( #ioGoHomePosition )
      Contact( #iHomePositionSensor )
      I_Contact( #ioManualGoWork )
      I_Contact( #ioAutoGoWork )
   END_RUNG wire#w5
   // the same network as SCL:
   #_w1 := #iRun AND #iEStop AND NOT #iError;
   #ioGoWorkPosition := #_w1 AND ((#iManualMode AND (#ioManualGoWork OR (#iManualOutputType AND #ioGoWorkPosition AND NOT #ioManualGoHome))) OR (#iAutoMode AND #ioAutoGoWork) OR (#ioGoWorkPosition AND #iWorkPositionSensor AND NOT #ioManualGoHome AND NOT #ioAutoGoHome)) AND #iGoWorkInterlock AND NOT #ioGoHomePosition;
   #ioGoHomePosition := #_w1 AND ((#iManualMode AND (#ioManualGoHome OR (#iManualOutputType AND #ioGoHomePosition AND NOT #ioManualGoWork))) OR (#iAutoMode AND #ioAutoGoHome) OR (#ioGoHomePosition AND #iHomePositionSensor AND NOT #ioManualGoWork AND NOT #ioAutoGoWork)) AND #iGoHomeInterlock AND NOT #ioGoWorkPosition;
END_REGION

REGION Network 5: Go_work_fault
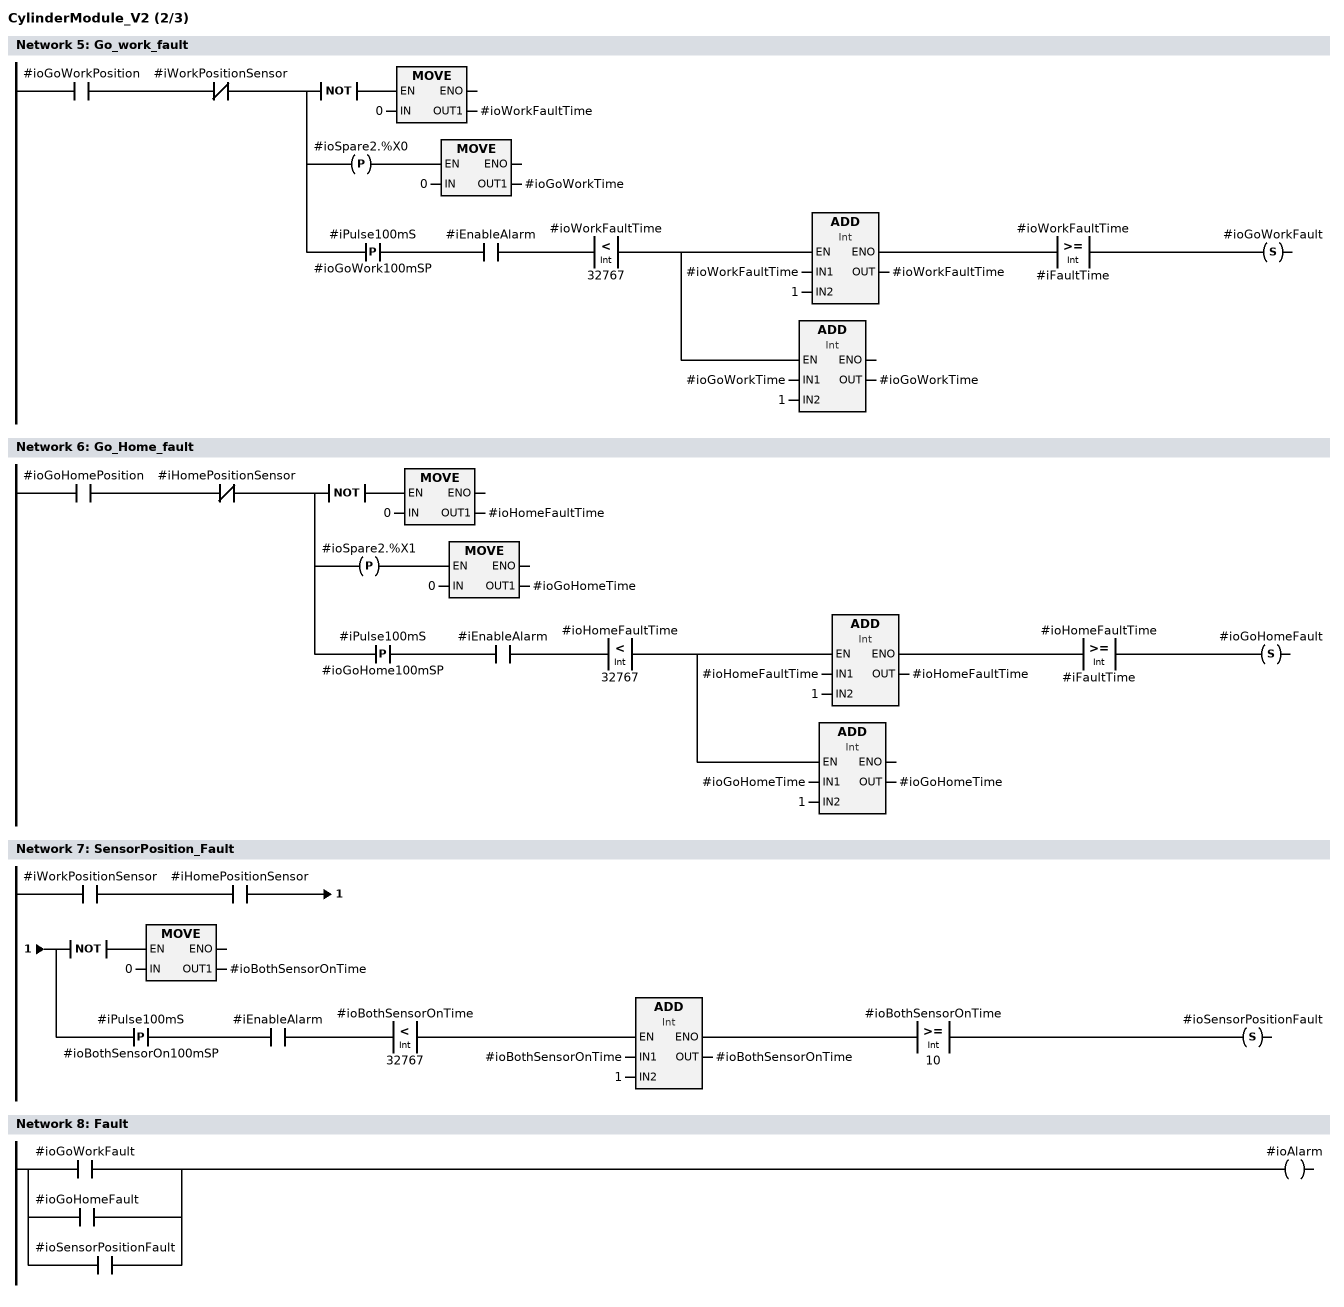
   RUNG wire#powerrail
      Contact( #ioGoWorkPosition )
      I_Contact( #iWorkPositionSensor )
      wire#w1
      Not()
      { S7_GenerateENO := "TRUE" } Move(in := 0, out1 => #ioWorkFaultTime)
   END_RUNG
   RUNG wire#w1
      P_Trig( #ioSpare2.%X0 )
      { S7_GenerateENO := "TRUE" } Move(in := 0, out1 => #ioGoWorkTime)
   END_RUNG
   RUNG wire#w1
      P_Contact(operand := #iPulse100mS, bit := #ioGoWork100mSP)
      Contact( #iEnableAlarm )
      { S7_Templates := "SrcType := Int" } LT_Contact(in1 := #ioWorkFaultTime, in2 := 32767)
      wire#w2
      { S7_Templates := "SrcType := Int"; S7_GenerateENO := "TRUE" } Add(in1 := #ioWorkFaultTime, in2 := 1, out => #ioWorkFaultTime)
      { S7_Templates := "SrcType := Int" } GE_Contact(in1 := #ioWorkFaultTime, in2 := #iFaultTime)
      S_Coil( #ioGoWorkFault )
   END_RUNG
   RUNG wire#w2
      { S7_Templates := "SrcType := Int"; S7_GenerateENO := "TRUE" } Add(in1 := #ioGoWorkTime, in2 := 1, out => #ioGoWorkTime)
   END_RUNG
   // the same network as SCL:
   // ENO of a box is taken as its EN; it also drops when the box reports an error
   #_w1 := #ioGoWorkPosition AND NOT #iWorkPositionSensor;
   IF NOT #_w1 THEN #ioWorkFaultTime := 0; END_IF;
   #_w2 := #_w1 AND NOT #ioSpare2.%X0;   // rising edge
   #ioSpare2.%X0 := #_w1;
   IF #_w2 THEN #ioGoWorkTime := 0; END_IF;
   #_w3 := #_w1 AND #iPulse100mS AND NOT #ioGoWork100mSP;   // rising edge of #iPulse100mS
   #ioGoWork100mSP := #iPulse100mS;
   #_w4 := #_w3 AND #iEnableAlarm AND (#ioWorkFaultTime < 32767);
   IF #_w4 THEN #ioWorkFaultTime := #ioWorkFaultTime + 1; END_IF;
   IF #_w4 AND (#ioWorkFaultTime >= #iFaultTime) THEN #ioGoWorkFault := TRUE; END_IF;
   IF #_w4 THEN #ioGoWorkTime := #ioGoWorkTime + 1; END_IF;
END_REGION

REGION Network 6: Go_Home_fault
   RUNG wire#powerrail
      Contact( #ioGoHomePosition )
      I_Contact( #iHomePositionSensor )
      wire#w1
      Not()
      { S7_GenerateENO := "TRUE" } Move(in := 0, out1 => #ioHomeFaultTime)
   END_RUNG
   RUNG wire#w1
      P_Trig( #ioSpare2.%X1 )
      { S7_GenerateENO := "TRUE" } Move(in := 0, out1 => #ioGoHomeTime)
   END_RUNG
   RUNG wire#w1
      P_Contact(operand := #iPulse100mS, bit := #ioGoHome100mSP)
      Contact( #iEnableAlarm )
      { S7_Templates := "SrcType := Int" } LT_Contact(in1 := #ioHomeFaultTime, in2 := 32767)
      wire#w2
      { S7_Templates := "SrcType := Int"; S7_GenerateENO := "TRUE" } Add(in1 := #ioHomeFaultTime, in2 := 1, out => #ioHomeFaultTime)
      { S7_Templates := "SrcType := Int" } GE_Contact(in1 := #ioHomeFaultTime, in2 := #iFaultTime)
      S_Coil( #ioGoHomeFault )
   END_RUNG
   RUNG wire#w2
      { S7_Templates := "SrcType := Int"; S7_GenerateENO := "TRUE" } Add(in1 := #ioGoHomeTime, in2 := 1, out => #ioGoHomeTime)
   END_RUNG
   // the same network as SCL:
   // ENO of a box is taken as its EN; it also drops when the box reports an error
   #_w1 := #ioGoHomePosition AND NOT #iHomePositionSensor;
   IF NOT #_w1 THEN #ioHomeFaultTime := 0; END_IF;
   #_w2 := #_w1 AND NOT #ioSpare2.%X1;   // rising edge
   #ioSpare2.%X1 := #_w1;
   IF #_w2 THEN #ioGoHomeTime := 0; END_IF;
   #_w3 := #_w1 AND #iPulse100mS AND NOT #ioGoHome100mSP;   // rising edge of #iPulse100mS
   #ioGoHome100mSP := #iPulse100mS;
   #_w4 := #_w3 AND #iEnableAlarm AND (#ioHomeFaultTime < 32767);
   IF #_w4 THEN #ioHomeFaultTime := #ioHomeFaultTime + 1; END_IF;
   IF #_w4 AND (#ioHomeFaultTime >= #iFaultTime) THEN #ioGoHomeFault := TRUE; END_IF;
   IF #_w4 THEN #ioGoHomeTime := #ioGoHomeTime + 1; END_IF;
END_REGION

REGION Network 7: SensorPosition_Fault
   RUNG wire#powerrail
      Contact( #iWorkPositionSensor )
      Contact( #iHomePositionSensor )
      wire#w1
      Not()
      { S7_GenerateENO := "TRUE" } Move(in := 0, out1 => #ioBothSensorOnTime)
   END_RUNG
   RUNG wire#w1
      P_Contact(operand := #iPulse100mS, bit := #ioBothSensorOn100mSP)
      Contact( #iEnableAlarm )
      { S7_Templates := "SrcType := Int" } LT_Contact(in1 := #ioBothSensorOnTime, in2 := 32767)
      { S7_Templates := "SrcType := Int"; S7_GenerateENO := "TRUE" } Add(in1 := #ioBothSensorOnTime, in2 := 1, out => #ioBothSensorOnTime)
      { S7_Templates := "SrcType := Int" } GE_Contact(in1 := #ioBothSensorOnTime, in2 := 10)
      S_Coil( #ioSensorPositionFault )
   END_RUNG
   // the same network as SCL:
   // ENO of a box is taken as its EN; it also drops when the box reports an error
   #_w1 := #iWorkPositionSensor AND #iHomePositionSensor;
   IF NOT #_w1 THEN #ioBothSensorOnTime := 0; END_IF;
   #_w2 := #_w1 AND #iPulse100mS AND NOT #ioBothSensorOn100mSP;   // rising edge of #iPulse100mS
   #ioBothSensorOn100mSP := #iPulse100mS;
   #_w3 := #_w2 AND #iEnableAlarm AND (#ioBothSensorOnTime < 32767);
   IF #_w3 THEN #ioBothSensorOnTime := #ioBothSensorOnTime + 1; END_IF;
   IF #_w3 AND (#ioBothSensorOnTime >= 10) THEN #ioSensorPositionFault := TRUE; END_IF;
END_REGION

REGION Network 8: Fault
   RUNG wire#powerrail
      Contact( #ioGoWorkFault )
      wire#w1
      Coil( #ioAlarm )
   END_RUNG
   RUNG wire#powerrail
      Contact( #ioGoHomeFault )
   END_RUNG wire#w1
   RUNG wire#powerrail
      Contact( #ioSensorPositionFault )
   END_RUNG wire#w1
   // the same network as SCL:
   #ioAlarm := #ioGoWorkFault OR #ioGoHomeFault OR #ioSensorPositionFault;
END_REGION

REGION Network 9: Reset fault
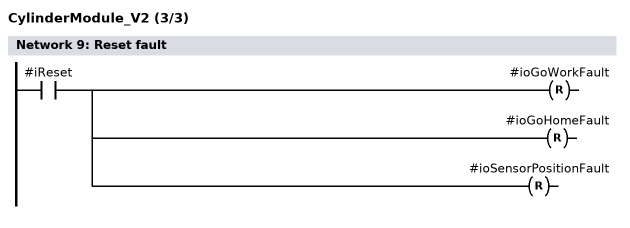
   RUNG wire#powerrail
      Contact( #iReset )
      wire#w1
      R_Coil( #ioGoWorkFault )
   END_RUNG
   RUNG wire#w1
      R_Coil( #ioGoHomeFault )
   END_RUNG
   RUNG wire#w1
      R_Coil( #ioSensorPositionFault )
   END_RUNG
   // the same network as SCL:
   IF #iReset THEN
       #ioGoWorkFault := FALSE;
       #ioGoHomeFault := FALSE;
       #ioSensorPositionFault := FALSE;
   END_IF;
END_REGION
END_FUNCTION

FUNCTION_BLOCK "MaterialGate"   // FB5210, LAD
{ S7_Optimized_Access := 'FALSE' }
// stored: AutoNumber false, SetENOAutomatically false
   VAR_INPUT
      iSysInface : "RCS_SysComInterface_V1";
      "iMaterialGate Opened Monitor" : Bool;   // 安全门打开状态监控
      "iMaterialGate Locked Monitor" : Bool;   // 安全门锁定状态监控
      i1s_Pulse : Bool;   // 1s脉冲信号
      "iMaterialGate AutoLock Timer" : Time := T#1s;   // 安全门自动模式下锁延时
      "iMaterialGate ManualLock Timer" : Time := T#60s;   // 安全门手动模式下锁定延时
   END_VAR
   VAR_OUTPUT
      "oMaterialGate LockedLamp" { ExternalAccessible := 'False'; ExternalVisible := 'False'; ExternalWritable := 'False'} : Bool;   // 安全门解锁输出状态
   END_VAR
   VAR_IN_OUT
      ioMaterialGateLock : Bool;   // 安全门锁定输出
      ioHMI_Interface : "SafetyGateUDT";
   END_VAR
   VAR
      "sMaterialafetyGate Timer" { S7_SetPoint := 'True'} : Array[1..5] of TON_TIME;
      sP_Trig : Array[1..10] of Bool;
      sN_Trig : Array[1..10] of Bool;
      "sMaterialGate UnlockRequest" { ExternalAccessible := 'False'; ExternalVisible := 'False'; ExternalWritable := 'False'} : Bool;   // 安全门开门请求标志位
      "sMaterialGate LockRequest" : Bool;
   END_VAR
   VAR_TEMP
      tAlyways_On : Bool;
      tAlyways_Off : Bool;
   END_VAR
   VAR_TEMP   // added for the SCL form of the ladder/FBD networks
      _w1 : Bool;
      _w2 : Bool;
      _w3 : Bool;
      _w4 : Bool;
      _w5 : Bool;
      _w6 : Bool;
      _w7 : Bool;
   END_VAR
BEGIN

REGION Network 1: #tAlyways_On
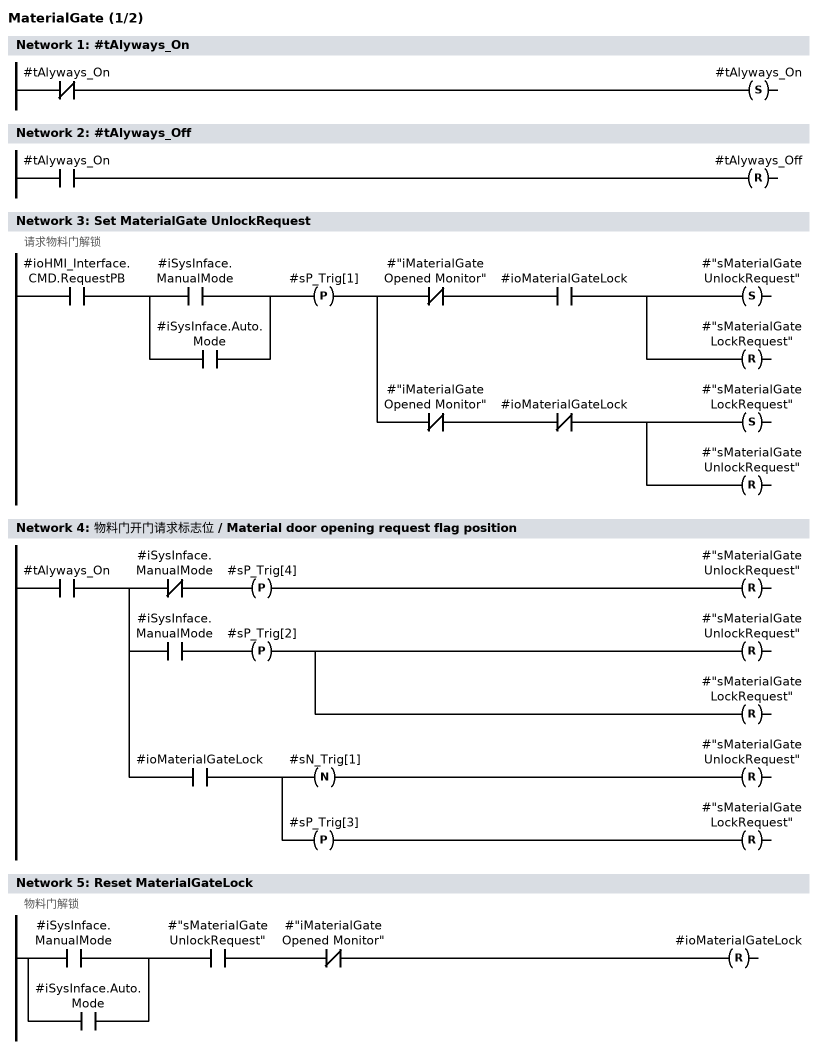
   RUNG wire#powerrail
      I_Contact( #tAlyways_On )
      S_Coil( #tAlyways_On )
   END_RUNG
   // the same network as SCL:
   IF NOT #tAlyways_On THEN #tAlyways_On := TRUE; END_IF;
END_REGION

REGION Network 2: #tAlyways_Off
   RUNG wire#powerrail
      Contact( #tAlyways_On )
      R_Coil( #tAlyways_Off )
   END_RUNG
   // the same network as SCL:
   IF #tAlyways_On THEN #tAlyways_Off := FALSE; END_IF;
END_REGION

REGION Network 3: Set MaterialGate UnlockRequest
   // 请求物料门解锁
   RUNG wire#powerrail
      Contact( #ioHMI_Interface.CMD.RequestPB )
      wire#w1
      Contact( #iSysInface.ManualMode )
      wire#w2
      P_Trig( #sP_Trig[1] )
      wire#w3
      I_Contact( #"iMaterialGate Opened Monitor" )
      Contact( #ioMaterialGateLock )
      wire#w4
      S_Coil( #"sMaterialGate UnlockRequest" )
   END_RUNG
   RUNG wire#w1
      Contact( #iSysInface.Auto.Mode )
   END_RUNG wire#w2
   RUNG wire#w4
      R_Coil( #"sMaterialGate LockRequest" )
   END_RUNG
   RUNG wire#w3
      I_Contact( #"iMaterialGate Opened Monitor" )
      I_Contact( #ioMaterialGateLock )
      wire#w5
      S_Coil( #"sMaterialGate LockRequest" )
   END_RUNG
   RUNG wire#w5
      R_Coil( #"sMaterialGate UnlockRequest" )
   END_RUNG
   // the same network as SCL:
   #_w1 := #ioHMI_Interface.CMD.RequestPB AND (#iSysInface.ManualMode OR #iSysInface.Auto.Mode);
   #_w2 := #_w1 AND NOT #sP_Trig[1];   // rising edge
   #sP_Trig[1] := #_w1;
   IF #_w2 AND NOT #"iMaterialGate Opened Monitor" AND #ioMaterialGateLock THEN
       #"sMaterialGate UnlockRequest" := TRUE;
       #"sMaterialGate LockRequest" := FALSE;
   END_IF;
   IF #_w2 AND NOT #"iMaterialGate Opened Monitor" AND NOT #ioMaterialGateLock THEN
       #"sMaterialGate LockRequest" := TRUE;
       #"sMaterialGate UnlockRequest" := FALSE;
   END_IF;
END_REGION

REGION Network 4: 物料门开门请求标志位 / Material door opening request flag position
   RUNG wire#powerrail
      Contact( #tAlyways_On )
      wire#w1
      I_Contact( #iSysInface.ManualMode )
      P_Trig( #sP_Trig[4] )
      R_Coil( #"sMaterialGate UnlockRequest" )
   END_RUNG
   RUNG wire#w1
      Contact( #iSysInface.ManualMode )
      P_Trig( #sP_Trig[2] )
      wire#w2
      R_Coil( #"sMaterialGate UnlockRequest" )
   END_RUNG
   RUNG wire#w2
      R_Coil( #"sMaterialGate LockRequest" )
   END_RUNG
   RUNG wire#w1
      Contact( #ioMaterialGateLock )
      wire#w3
      N_Trig( #sN_Trig[1] )
      R_Coil( #"sMaterialGate UnlockRequest" )
   END_RUNG
   RUNG wire#w3
      P_Trig( #sP_Trig[3] )
      R_Coil( #"sMaterialGate LockRequest" )
   END_RUNG
   // the same network as SCL:
   #_w1 := #tAlyways_On AND NOT #iSysInface.ManualMode;
   #_w2 := #_w1 AND NOT #sP_Trig[4];   // rising edge
   #sP_Trig[4] := #_w1;
   IF #_w2 THEN #"sMaterialGate UnlockRequest" := FALSE; END_IF;
   #_w3 := #tAlyways_On AND #iSysInface.ManualMode;
   #_w4 := #_w3 AND NOT #sP_Trig[2];   // rising edge
   #sP_Trig[2] := #_w3;
   IF #_w4 THEN
       #"sMaterialGate UnlockRequest" := FALSE;
       #"sMaterialGate LockRequest" := FALSE;
   END_IF;
   #_w5 := #tAlyways_On AND #ioMaterialGateLock;
   #_w6 := NOT #_w5 AND #sN_Trig[1];   // falling edge
   #sN_Trig[1] := #_w5;
   IF #_w6 THEN #"sMaterialGate UnlockRequest" := FALSE; END_IF;
   #_w7 := #_w5 AND NOT #sP_Trig[3];   // rising edge
   #sP_Trig[3] := #_w5;
   IF #_w7 THEN #"sMaterialGate LockRequest" := FALSE; END_IF;
END_REGION

REGION Network 5: Reset MaterialGateLock
   // 物料门解锁
   RUNG wire#powerrail
      Contact( #iSysInface.ManualMode )
      wire#w1
      Contact( #"sMaterialGate UnlockRequest" )
      I_Contact( #"iMaterialGate Opened Monitor" )
      R_Coil( #ioMaterialGateLock )
   END_RUNG
   RUNG wire#powerrail
      Contact( #iSysInface.Auto.Mode )
   END_RUNG wire#w1
   // the same network as SCL:
   IF (#iSysInface.ManualMode OR #iSysInface.Auto.Mode) AND #"sMaterialGate UnlockRequest" AND NOT #"iMaterialGate Opened Monitor" THEN
       #ioMaterialGateLock := FALSE;
   END_IF;
END_REGION

REGION Network 6: Set MaterialGate Lock
   // 物料门锁定
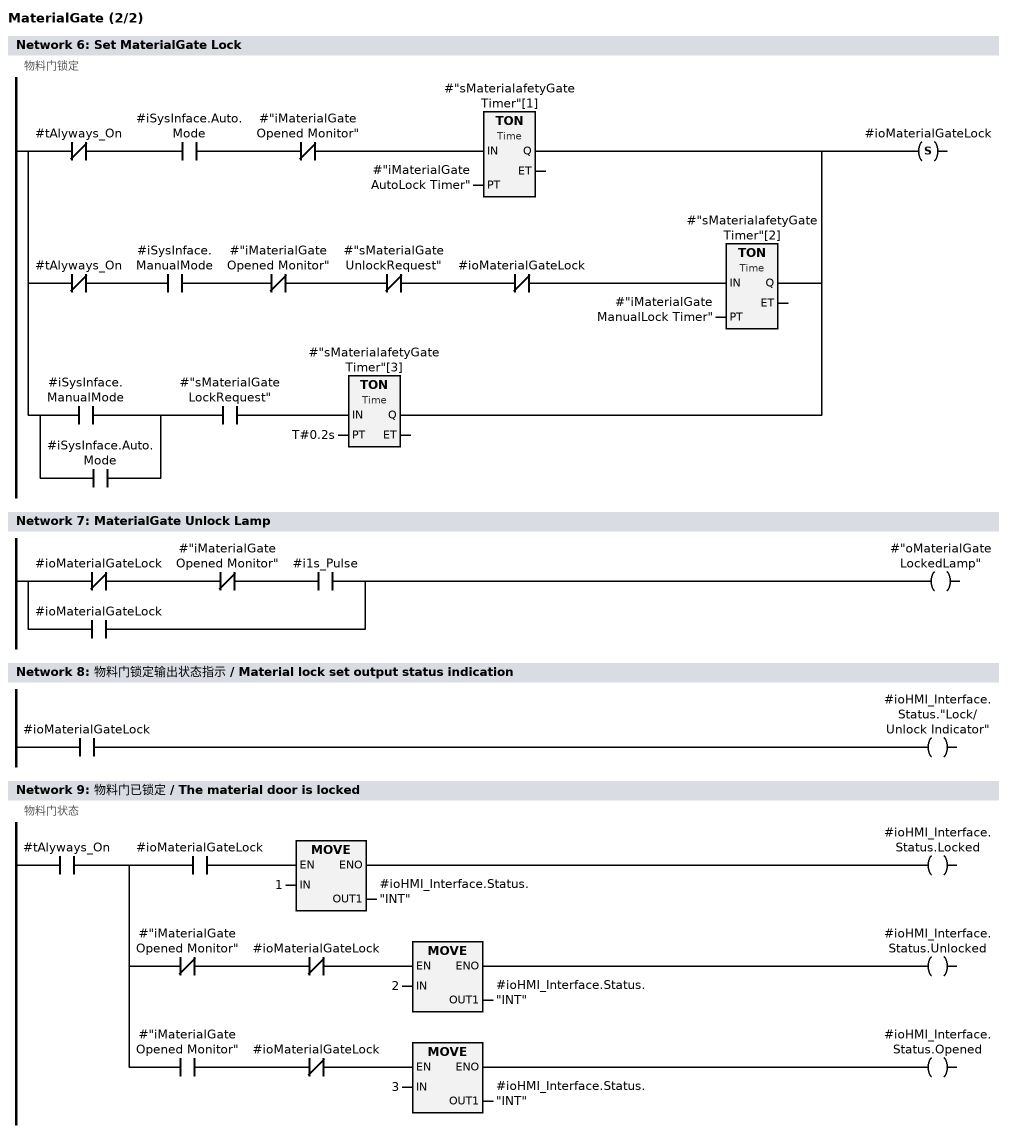
   RUNG wire#powerrail
      I_Contact( #tAlyways_On )
      Contact( #iSysInface.Auto.Mode )
      I_Contact( #"iMaterialGate Opened Monitor" )
      { S7_Templates := "time_type := Time" } #"sMaterialafetyGate Timer"[1].TON(pt := #"iMaterialGate AutoLock Timer", et =>)
      wire#w1
      S_Coil( #ioMaterialGateLock )
   END_RUNG
   RUNG wire#powerrail
      I_Contact( #tAlyways_On )
      Contact( #iSysInface.ManualMode )
      I_Contact( #"iMaterialGate Opened Monitor" )
      I_Contact( #"sMaterialGate UnlockRequest" )
      I_Contact( #ioMaterialGateLock )
      { S7_Templates := "time_type := Time" } #"sMaterialafetyGate Timer"[2].TON(pt := #"iMaterialGate ManualLock Timer", et =>)
   END_RUNG wire#w1
   RUNG wire#powerrail
      Contact( #iSysInface.ManualMode )
      wire#w2
      Contact( #"sMaterialGate LockRequest" )
      { S7_Templates := "time_type := Time" } #"sMaterialafetyGate Timer"[3].TON(pt := T#0.2s, et =>)
   END_RUNG wire#w1
   RUNG wire#powerrail
      Contact( #iSysInface.Auto.Mode )
   END_RUNG wire#w2
   // the same network as SCL:
   #"sMaterialafetyGate Timer"[1].TON(IN := NOT #tAlyways_On AND #iSysInface.Auto.Mode AND NOT #"iMaterialGate Opened Monitor",
                           PT := #"iMaterialGate AutoLock Timer");
   #_w1 := #"sMaterialafetyGate Timer"[1].Q;
   #"sMaterialafetyGate Timer"[2].TON(IN := NOT #tAlyways_On AND #iSysInface.ManualMode AND NOT #"iMaterialGate Opened Monitor" AND NOT #"sMaterialGate UnlockRequest" AND NOT #ioMaterialGateLock,
                           PT := #"iMaterialGate ManualLock Timer");
   #_w2 := #"sMaterialafetyGate Timer"[2].Q;
   #"sMaterialafetyGate Timer"[3].TON(IN := (#iSysInface.ManualMode OR #iSysInface.Auto.Mode) AND #"sMaterialGate LockRequest",
                           PT := T#0.2s);
   IF #_w1 OR #_w2 OR #"sMaterialafetyGate Timer"[3].Q THEN #ioMaterialGateLock := TRUE; END_IF;
END_REGION

REGION Network 7: MaterialGate Unlock Lamp
   RUNG wire#powerrail
      I_Contact( #ioMaterialGateLock )
      I_Contact( #"iMaterialGate Opened Monitor" )
      Contact( #i1s_Pulse )
      wire#w1
      Coil( #"oMaterialGate LockedLamp" )
   END_RUNG
   RUNG wire#powerrail
      Contact( #ioMaterialGateLock )
   END_RUNG wire#w1
   // the same network as SCL:
   #"oMaterialGate LockedLamp" := (NOT #ioMaterialGateLock AND NOT #"iMaterialGate Opened Monitor" AND #i1s_Pulse) OR #ioMaterialGateLock;
END_REGION

REGION Network 8: 物料门锁定输出状态指示 / Material lock set output status indication
   RUNG wire#powerrail
      Contact( #ioMaterialGateLock )
      Coil( #ioHMI_Interface.Status."Lock/Unlock Indicator" )
   END_RUNG
   // the same network as SCL:
   #ioHMI_Interface.Status."Lock/Unlock Indicator" := #ioMaterialGateLock;
END_REGION

REGION Network 9: 物料门已锁定 / The material door is locked
   // 物料门状态
   RUNG wire#powerrail
      Contact( #tAlyways_On )
      wire#w1
      Contact( #ioMaterialGateLock )
      Move(in := 1, out1 => #ioHMI_Interface.Status."INT")
      Coil( #ioHMI_Interface.Status.Locked )
   END_RUNG
   RUNG wire#w1
      I_Contact( #"iMaterialGate Opened Monitor" )
      I_Contact( #ioMaterialGateLock )
      Move(in := 2, out1 => #ioHMI_Interface.Status."INT")
      Coil( #ioHMI_Interface.Status.Unlocked )
   END_RUNG
   RUNG wire#w1
      Contact( #"iMaterialGate Opened Monitor" )
      I_Contact( #ioMaterialGateLock )
      Move(in := 3, out1 => #ioHMI_Interface.Status."INT")
      Coil( #ioHMI_Interface.Status.Opened )
   END_RUNG
   // the same network as SCL:
   #_w1 := #tAlyways_On AND #ioMaterialGateLock;
   IF #_w1 THEN #ioHMI_Interface.Status."INT" := 1; END_IF;
   #ioHMI_Interface.Status.Locked := #_w1;
   #_w2 := #tAlyways_On AND NOT #"iMaterialGate Opened Monitor" AND NOT #ioMaterialGateLock;
   IF #_w2 THEN #ioHMI_Interface.Status."INT" := 2; END_IF;
   #ioHMI_Interface.Status.Unlocked := #_w2;
   #_w3 := #tAlyways_On AND #"iMaterialGate Opened Monitor" AND NOT #ioMaterialGateLock;
   IF #_w3 THEN #ioHMI_Interface.Status."INT" := 3; END_IF;
   #ioHMI_Interface.Status.Opened := #_w3;
END_REGION
END_FUNCTION_BLOCK

FUNCTION_BLOCK "PartDataManage"   // FB2, SCL
{ S7_Optimized_Access := 'TRUE' }
// stored: MemoryReserve 100, SetENOAutomatically false
   VAR_INPUT
      iReset : Bool;   // 复位
      iScannerTrigger : Bool;   // 扫码枪触发
      iStringRecived : String;   // 扫码枪接收到的物料码
      iMaterialType : String;   // 设定的物料型号
      iSaveToBuffer : Bool;   // 触发将物料信息存储到缓存
      iCodeType : Bool;   // 物料码类型：0，批次码，1，单件码
      iDecrementCnt : DInt := 1;   // 每次的用量
      iDecrementTrigger : Bool;   // 触发信号
      iBufferBoxes : Int := 1;   // 允许缓存的数量,最小为1，最大5
   END_VAR
   VAR_IN_OUT
      ioMaterialActive : Bool;   // 物料比对成功
      io_MaterialManage : "PartData_UDT";
   END_VAR
   VAR
      NO : Array[0..6] of Int;
      sString_MId : String;
      sKeyChar : Char := '#';
      Puls : Array[0..20] of Bool;
      R_TRIG_MaterialActive { S7_SetPoint := 'True'} : R_TRIG;
      R_TRIG_ScannerTrigger { S7_SetPoint := 'True'} : R_TRIG;
      IEC_Timer_MaterialActive { S7_SetPoint := 'True'} : TON_TIME;
      R_TRIG_DecrementTrigger { S7_SetPoint := 'True'} : R_TRIG;
      "R_TRIG_PartQuality+1" { S7_SetPoint := 'True'} : R_TRIG;
      "R_TRIG_PartQuality-1" { S7_SetPoint := 'True'} : R_TRIG;
      R_TRIG_ClearCurrentBox { S7_SetPoint := 'True'} : R_TRIG;
      R_TRIG_ClearAllBox { S7_SetPoint := 'True'} : R_TRIG;
      R_TRIG_SaveToBuffer { S7_SetPoint := 'True'} : R_TRIG;
      Timer_PartQualityAckPB { S7_SetPoint := 'True'} : TON_TIME;
   END_VAR
   VAR_TEMP
      tMaterialTypePos : Int;   // 设定物料码在接收码中的位置
      tLenString : Int;
      BufferIndex : Int;
      "BufferIndex+1" : Int;
      "BufferBoxes-1" : Int;
   END_VAR
BEGIN

   REGION Comment
       //本功能块针对豫北物料编码规则编写，其他项目或规则不宜直接引用：
       //本物料针对手持扫码枪需要扫多个物料的情况，
       //针对物料分为两种：
       //一：单件扫码，物料具有独立标识码，需要将变量  iCodeType  赋 true
       //同时，无需关注其他物料码解析，缓存等功能，
       //只使用    #iStringRecived / #ioMaterialActive 等变量，供程序判断扫码结果和获取物料码使用；
       //不需要配合使用HMI面板
       //二：物料为批次码，需要根据实际情况，设定缓存数量 #iBufferBoxes
       //同时根据需要创建使用HMI面板  
   END_REGION

   REGION 物料比对成功

       #R_TRIG_ScannerTrigger(CLK := #iScannerTrigger);

       #tMaterialTypePos := FIND(IN1 := #iStringRecived, IN2 := #iMaterialType);

       IF #R_TRIG_ScannerTrigger.Q AND #tMaterialTypePos <> 0 THEN
           #ioMaterialActive := 1;
       END_IF;
       //上升沿信号
       #R_TRIG_MaterialActive(CLK := #ioMaterialActive);

       //延时复位
       //
       #IEC_Timer_MaterialActive(IN := #ioMaterialActive,
                                 PT := T#300ms);

       IF #IEC_Timer_MaterialActive.Q THEN
           #ioMaterialActive := 0;
       END_IF;


   END_REGION

   REGION Recive Part Data Analysis

       IF #R_TRIG_MaterialActive.Q AND NOT #iCodeType THEN

           //PartCode
           #io_MaterialManage.PartBoxDataRecive.PartCode := #iStringRecived;
           #io_MaterialManage.PartBoxDataRecive.PartCode_Len := LEN(#io_MaterialManage.PartBoxDataRecive.PartCode);


           //SupplierID
           #NO[0] := FIND(IN1 := #iStringRecived, IN2 := #sKeyChar);
           #NO[1] := #NO[0] - 1;
           #io_MaterialManage.PartBoxDataRecive.SupplierID := LEFT(IN := #iStringRecived, L := #NO[1]);

           //MaterialType
           #tLenString := #io_MaterialManage.PartBoxDataRecive.PartCode_Len - #NO[0];
           #sString_MId := RIGHT_STRING(IN := #iStringRecived, L := #tLenString);
           #NO[0] := FIND(IN1 := #sString_MId, IN2 := #sKeyChar);
           #NO[2] := #NO[0] - 1;
           #io_MaterialManage.PartBoxDataRecive.MaterialType := LEFT(IN := #sString_MId, L := #NO[2]);

           //PO_ID
           //
           #tLenString := #tLenString - #NO[0];
           #sString_MId := RIGHT_STRING(IN := #sString_MId, L := #tLenString);
           #NO[0] := FIND(IN1 := #sString_MId, IN2 := #sKeyChar);
           #NO[3] := #NO[0] - 1;
           #io_MaterialManage.PartBoxDataRecive.PO_ID := LEFT(IN := #sString_MId, L := #NO[3]);

           //BatchID

           #tLenString := #tLenString - #NO[0];
           #sString_MId := RIGHT_STRING(IN := #sString_MId, L := #tLenString);
           #NO[0] := FIND(IN1 := #sString_MId, IN2 := #sKeyChar);
           #NO[4] := #NO[0] - 1;
           #io_MaterialManage.PartBoxDataRecive.BatchID := LEFT(IN := #sString_MId, L := #NO[4]);

           //Quality

           #tLenString := #tLenString - #NO[0];
           #sString_MId := RIGHT_STRING(IN := #sString_MId, L := #tLenString);
           #NO[0] := FIND(IN1 := #sString_MId, IN2 := #sKeyChar);
           #NO[5] := #NO[0] - 1;
           #io_MaterialManage.PartBoxDataRecive.Quality := LEFT(IN := #sString_MId, L := #NO[5]);

           //Cartons
           //
           #tLenString := #tLenString - #NO[0];
           #sString_MId := RIGHT_STRING(IN := #sString_MId, L := #tLenString);
           #io_MaterialManage.PartBoxDataRecive.Cartons := #sString_MId;

       END_IF;
   END_REGION

   REGION Waring
       //物料码已使用，扫码无效   
       IF #ioMaterialActive AND NOT #iCodeType THEN
           IF #io_MaterialManage.PartBoxDataRecive.PartCode = #io_MaterialManage.PartBoxData[1].PartCode
               OR #io_MaterialManage.PartBoxDataRecive.PartCode = #io_MaterialManage.PartBoxData[2].PartCode
               OR #io_MaterialManage.PartBoxDataRecive.PartCode = #io_MaterialManage.PartBoxData[3].PartCode
               OR #io_MaterialManage.PartBoxDataRecive.PartCode = #io_MaterialManage.PartBoxData[4].PartCode
               OR #io_MaterialManage.PartBoxDataRecive.PartCode = #io_MaterialManage.PartBoxData[5].PartCode THEN

               #io_MaterialManage.PartDataHMI.Waring.ScannCodeInvalid := 1;

           END_IF;

       END_IF;


       //物料缓存已满，无法保存
       IF #ioMaterialActive
           AND #io_MaterialManage.PartBoxData[#iBufferBoxes] <> #io_MaterialManage.PartBoxDataNull THEN
           #io_MaterialManage.PartDataHMI.Waring.BufferBoxFull := 1;

       END_IF;
       //物料不足，请及时添加

       IF #io_MaterialManage.PartDataHMI.PartQuality <= #iDecrementCnt THEN
           #io_MaterialManage.PartDataHMI.Waring.Insufficient := 1;

       END_IF;



       IF #iReset THEN

           #io_MaterialManage.PartDataHMI.Waring.Insufficient := 0;
           #io_MaterialManage.PartDataHMI.Waring.BufferBoxFull := 0;
           #io_MaterialManage.PartDataHMI.Waring.ScannCodeInvalid := 0;

       END_IF;

   END_REGION

   REGION Part Data Load LOOP
       IF NOT #iCodeType THEN

           IF #io_MaterialManage.PartDataHMI.PartQuality < #iDecrementCnt THEN

               #io_MaterialManage.PartBoxData[0] := #io_MaterialManage.PartBoxData[1];

               #io_MaterialManage.PartDataHMI.PartQuality := STRING_TO_DINT(IN := #io_MaterialManage.PartBoxData[0].Quality);


               #io_MaterialManage.PartBoxData[1] := #io_MaterialManage.PartBoxDataNull;

           END_IF;


           IF #iBufferBoxes > 1 THEN
               #BufferIndex := 1;
               #"BufferBoxes-1" := #iBufferBoxes - 1;
               FOR #BufferIndex := 1 TO #iBufferBoxes - 1 DO

                   #"BufferIndex+1" := #BufferIndex + 1;

                   IF #io_MaterialManage.PartBoxData[#BufferIndex] = #io_MaterialManage.PartBoxDataNull THEN

                       #io_MaterialManage.PartBoxData[#BufferIndex] := #io_MaterialManage.PartBoxData[#"BufferIndex+1"];

                       #io_MaterialManage.PartBoxData[#"BufferIndex+1"] := #io_MaterialManage.PartBoxDataNull;
                   END_IF;

               END_FOR;

           END_IF;

       END_IF;


       #R_TRIG_SaveToBuffer(CLK:=#iSaveToBuffer);



       IF #R_TRIG_SaveToBuffer.Q AND NOT #iCodeType AND NOT #io_MaterialManage.PartDataHMI.Waring.ScannCodeInvalid
           AND #io_MaterialManage.PartBoxData[#iBufferBoxes] = #io_MaterialManage.PartBoxDataNull THEN

           #io_MaterialManage.PartBoxData[#iBufferBoxes] := #io_MaterialManage.PartBoxDataRecive;

           #io_MaterialManage.PartBoxDataRecive := #io_MaterialManage.PartBoxDataNull;
       END_IF;
   END_REGION

   REGION Part quality 
       //Part quality Decrement
       #R_TRIG_DecrementTrigger(CLK := #iDecrementTrigger);
       IF #R_TRIG_DecrementTrigger.Q THEN
           #io_MaterialManage.PartDataHMI.PartQuality := #io_MaterialManage.PartDataHMI.PartQuality - #iDecrementCnt;
       END_IF;

      // Part quality Adjust
       #"R_TRIG_PartQuality+1"(CLK:=#io_MaterialManage.PartDataHMI.CMD."PartQuality+1");
       #"R_TRIG_PartQuality-1"(CLK:=#io_MaterialManage.PartDataHMI.CMD."PartQuality-1");

       IF #"R_TRIG_PartQuality+1".Q THEN
           #io_MaterialManage.PartDataHMI.PartQuality :=#io_MaterialManage.PartDataHMI.PartQuality + 1;
       END_IF;
       IF #"R_TRIG_PartQuality-1".Q THEN
           #io_MaterialManage.PartDataHMI.PartQuality := #io_MaterialManage.PartDataHMI.PartQuality - 1;

       END_IF;

       // Part quality Set By Operator
       #Timer_PartQualityAckPB(IN:=#io_MaterialManage.PartDataHMI.CMD.PartQualityAck,
                               PT:=t#2s);

       IF #Timer_PartQualityAckPB.Q THEN

           #io_MaterialManage.PartDataHMI.PartQuality := #io_MaterialManage.PartDataHMI.PartQualitySet;
       END_IF;




       // Part Data Clear
       #R_TRIG_ClearCurrentBox(CLK := #io_MaterialManage.PartDataHMI.CMD.ClearCurrentBox);
       #R_TRIG_ClearAllBox(CLK := #io_MaterialManage.PartDataHMI.CMD.ClearAllBox);

       IF #R_TRIG_ClearCurrentBox.Q THEN
           #io_MaterialManage.PartBoxData[0] := #io_MaterialManage.PartBoxDataNull;

       END_IF;

       IF #R_TRIG_ClearAllBox.Q THEN

           #BufferIndex := 0;
           FOR #BufferIndex := 0 TO 20 DO
               #io_MaterialManage.PartBoxData[#BufferIndex] := #io_MaterialManage.PartBoxDataNull;
           END_FOR;
       END_IF;

   END_REGION


   REGION PartData Dispaly
       #io_MaterialManage.PartDataHMI.PartDataDispaly := #io_MaterialManage.PartBoxData[#io_MaterialManage.PartDataHMI.BoxDisplayID];
   END_REGION
END_FUNCTION_BLOCK

FUNCTION_BLOCK "FB_Stopper"   // FB4001, LAD
{ S7_Optimized_Access := 'FALSE' }
// stored: AutoNumber false, SetENOAutomatically false
   VAR_INPUT
      iSysInface : "RCS_SysComInterface_V1";
      iSensor : Bool;   // 本站托盘到位
      iNextSensor : Bool;   // 后站托盘到位
      iNextValve : Bool;   // 后站挡停输出
      iPresentDwell : Time := T#0.3s;   // 本站到位传感器延时
      iNextEmptyDwell : Time := T#10s;   // 后站托盘到位传感器延时
      iReleaseClear : Bool;   // 托盘释放允许
      iReleaseDwell : Time := T#1s;   // 托盘已流出延时
      iReleaseFaultTimer : Time := T#1s;   // 托盘流出超时延时
      iReachFaultTimer : Time := T#5s;   // 托盘流入后站超时延时
   END_VAR
   VAR_OUTPUT
      oValve : Bool;   // 本站挡停输出
      oReleaseCompleted : Bool;   // 释放完成
      oReleaseFault : Bool;   // 托盘流走超时
      oReachFault : Bool;   // 后站托盘接收超时
      oNotClear : Bool;   // 手动释放中
   END_VAR
   VAR_IN_OUT
      io_Dev : "ST_Stopper";
   END_VAR
   VAR
      Stopper : Struct
         Sensor : Bool;
         Valve : Bool;
         NextSensor : Bool;
         NextValve : Bool;
         NextFullSensor : Bool;
         PresentDwell : TON_TIME;
         NextEmptyDwell : TON_TIME;
         NextFullDwell : TON_TIME;
         ReleaseClear : Bool;
         ReleaseMemory : Bool;
         ReleaseDwell : TON_TIME;
         ReleasePB : Bool;
         NotClear : Bool;
         NextEmptyMemory : Bool;
         ReleaseCompleted : Bool;
         ReleaseFaultTimer : TON_TIME;
         ReachFaultTimer : TON_TIME;
      END_STRUCT;
   END_VAR
BEGIN

REGION Network 1: 输入输出映射 / Input output map
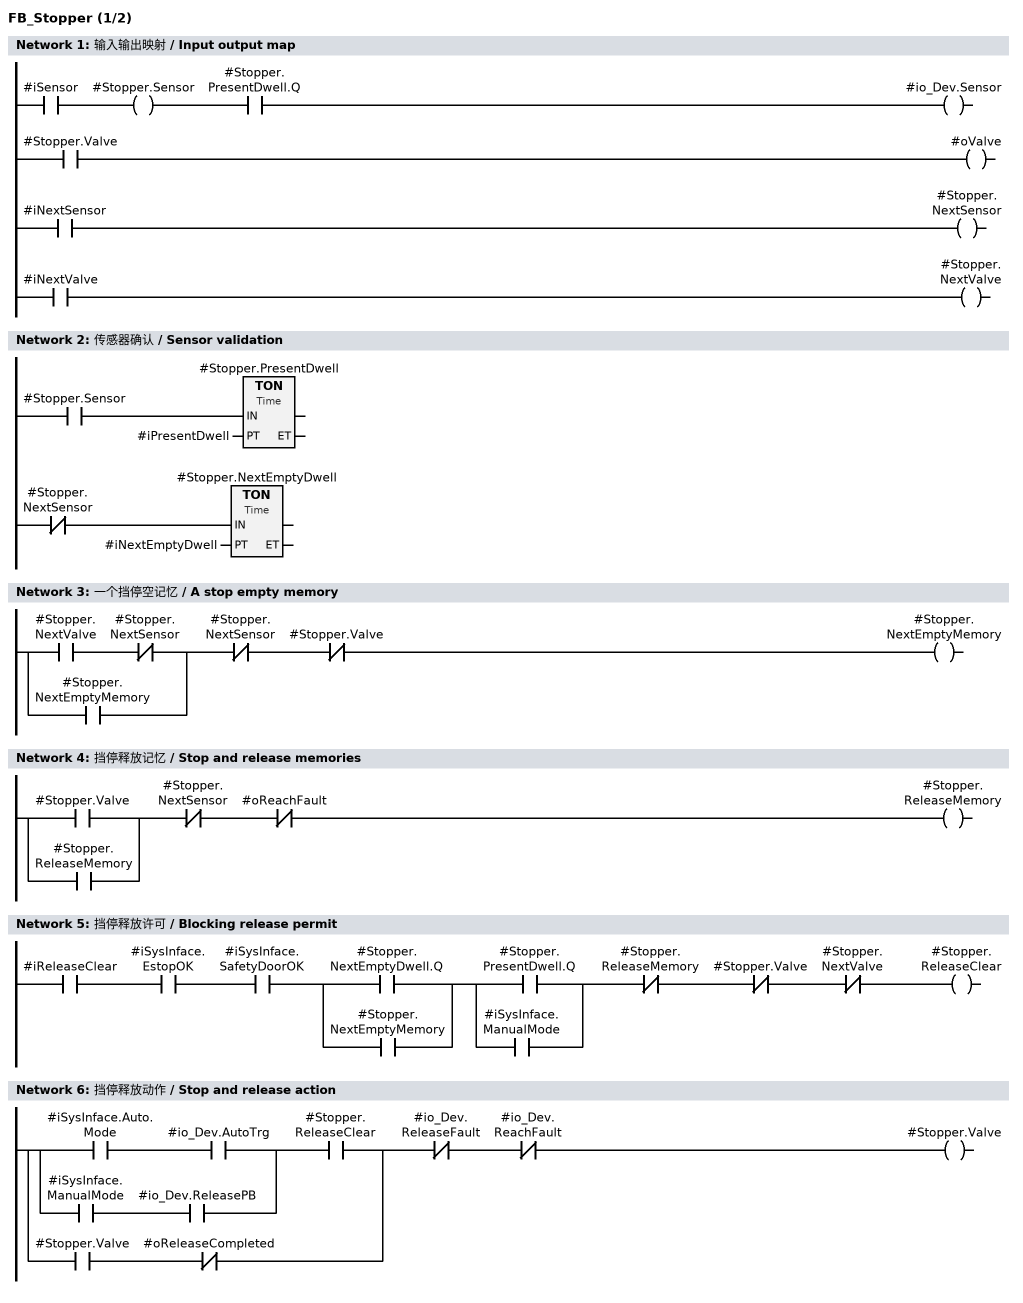
   RUNG wire#powerrail
      Contact( #iSensor )
      Coil( #Stopper.Sensor )
      Contact( #Stopper.PresentDwell.Q )
      Coil( #io_Dev.Sensor )
   END_RUNG
   RUNG wire#powerrail
      Contact( #Stopper.Valve )
      Coil( #oValve )
   END_RUNG
   RUNG wire#powerrail
      Contact( #iNextSensor )
      Coil( #Stopper.NextSensor )
   END_RUNG
   RUNG wire#powerrail
      Contact( #iNextValve )
      Coil( #Stopper.NextValve )
   END_RUNG
   // the same network as SCL:
   #Stopper.Sensor := #iSensor;
   #io_Dev.Sensor := #iSensor AND #Stopper.PresentDwell.Q;
   #oValve := #Stopper.Valve;
   #Stopper.NextSensor := #iNextSensor;
   #Stopper.NextValve := #iNextValve;
END_REGION

REGION Network 2: 传感器确认 / Sensor validation
   RUNG wire#powerrail
      Contact( #Stopper.Sensor )
      { S7_Templates := "time_type := Time" } #Stopper.PresentDwell.TON(pt := #iPresentDwell, et =>)
   END_RUNG
   RUNG wire#powerrail
      I_Contact( #Stopper.NextSensor )
      { S7_Templates := "time_type := Time" } #Stopper.NextEmptyDwell.TON(pt := #iNextEmptyDwell, et =>)
   END_RUNG
   // the same network as SCL:
   #Stopper.PresentDwell.TON(IN := #Stopper.Sensor, PT := #iPresentDwell);
   #Stopper.NextEmptyDwell.TON(IN := NOT #Stopper.NextSensor, PT := #iNextEmptyDwell);
END_REGION

REGION Network 3: 一个挡停空记忆 / A stop empty memory
   RUNG wire#powerrail
      Contact( #Stopper.NextValve )
      I_Contact( #Stopper.NextSensor )
      wire#w1
      I_Contact( #Stopper.NextSensor )
      I_Contact( #Stopper.Valve )
      Coil( #Stopper.NextEmptyMemory )
   END_RUNG
   RUNG wire#powerrail
      Contact( #Stopper.NextEmptyMemory )
   END_RUNG wire#w1
   // the same network as SCL:
   #Stopper.NextEmptyMemory := ((#Stopper.NextValve AND NOT #Stopper.NextSensor) OR #Stopper.NextEmptyMemory) AND NOT #Stopper.NextSensor AND NOT #Stopper.Valve;
END_REGION

REGION Network 4: 挡停释放记忆 / Stop and release memories
   RUNG wire#powerrail
      Contact( #Stopper.Valve )
      wire#w1
      I_Contact( #Stopper.NextSensor )
      I_Contact( #oReachFault )
      Coil( #Stopper.ReleaseMemory )
   END_RUNG
   RUNG wire#powerrail
      Contact( #Stopper.ReleaseMemory )
   END_RUNG wire#w1
   // the same network as SCL:
   #Stopper.ReleaseMemory := (#Stopper.Valve OR #Stopper.ReleaseMemory) AND NOT #Stopper.NextSensor AND NOT #oReachFault;
END_REGION

REGION Network 5: 挡停释放许可 / Blocking release permit
   RUNG wire#powerrail
      Contact( #iReleaseClear )
      Contact( #iSysInface.EstopOK )
      Contact( #iSysInface.SafetyDoorOK )
      wire#w1
      Contact( #Stopper.NextEmptyDwell.Q )
      wire#w2
      Contact( #Stopper.PresentDwell.Q )
      wire#w3
      I_Contact( #Stopper.ReleaseMemory )
      I_Contact( #Stopper.Valve )
      I_Contact( #Stopper.NextValve )
      Coil( #Stopper.ReleaseClear )
   END_RUNG
   RUNG wire#w1
      Contact( #Stopper.NextEmptyMemory )
   END_RUNG wire#w2
   RUNG wire#w2
      Contact( #iSysInface.ManualMode )
   END_RUNG wire#w3
   // the same network as SCL:
   #Stopper.ReleaseClear := #iReleaseClear AND #iSysInface.EstopOK AND #iSysInface.SafetyDoorOK AND (#Stopper.NextEmptyDwell.Q OR #Stopper.NextEmptyMemory) AND (#Stopper.PresentDwell.Q OR #iSysInface.ManualMode) AND NOT #Stopper.ReleaseMemory AND NOT #Stopper.Valve AND NOT #Stopper.NextValve;
END_REGION

REGION Network 6: 挡停释放动作 / Stop and release action
   RUNG wire#powerrail
      Contact( #iSysInface.Auto.Mode )
      Contact( #io_Dev.AutoTrg )
      wire#w1
      Contact( #Stopper.ReleaseClear )
      wire#w2
      I_Contact( #io_Dev.ReleaseFault )
      I_Contact( #io_Dev.ReachFault )
      Coil( #Stopper.Valve )
   END_RUNG
   RUNG wire#powerrail
      Contact( #iSysInface.ManualMode )
      Contact( #io_Dev.ReleasePB )
   END_RUNG wire#w1
   RUNG wire#powerrail
      Contact( #Stopper.Valve )
      I_Contact( #oReleaseCompleted )
   END_RUNG wire#w2
   // the same network as SCL:
   #Stopper.Valve := ((((#iSysInface.Auto.Mode AND #io_Dev.AutoTrg) OR (#iSysInface.ManualMode AND #io_Dev.ReleasePB)) AND #Stopper.ReleaseClear) OR (#Stopper.Valve AND NOT #oReleaseCompleted)) AND NOT #io_Dev.ReleaseFault AND NOT #io_Dev.ReachFault;
END_REGION

REGION Network 7: 释放完成信号 / Release completion signal
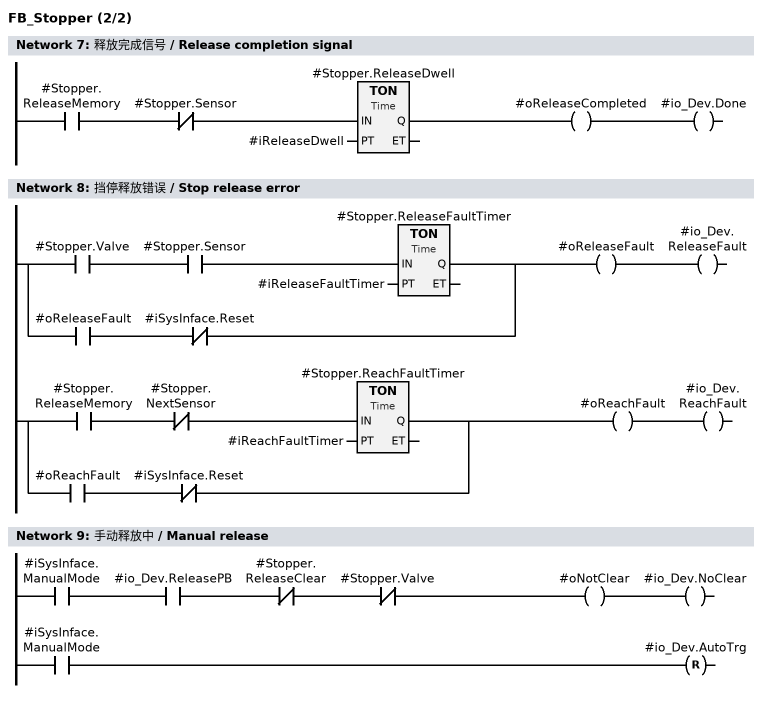
   RUNG wire#powerrail
      Contact( #Stopper.ReleaseMemory )
      I_Contact( #Stopper.Sensor )
      { S7_Templates := "time_type := Time" } #Stopper.ReleaseDwell.TON(pt := #iReleaseDwell, et =>)
      Coil( #oReleaseCompleted )
      Coil( #io_Dev.Done )
   END_RUNG
   // the same network as SCL:
   #Stopper.ReleaseDwell.TON(IN := #Stopper.ReleaseMemory AND NOT #Stopper.Sensor, PT := #iReleaseDwell);
   #oReleaseCompleted := #Stopper.ReleaseDwell.Q;
   #io_Dev.Done := #Stopper.ReleaseDwell.Q;
END_REGION

REGION Network 8: 挡停释放错误 / Stop release error
   RUNG wire#powerrail
      Contact( #Stopper.Valve )
      Contact( #Stopper.Sensor )
      { S7_Templates := "time_type := Time" } #Stopper.ReleaseFaultTimer.TON(pt := #iReleaseFaultTimer, et =>)
      wire#w1
      Coil( #oReleaseFault )
      Coil( #io_Dev.ReleaseFault )
   END_RUNG
   RUNG wire#powerrail
      Contact( #oReleaseFault )
      I_Contact( #iSysInface.Reset )
   END_RUNG wire#w1
   RUNG wire#powerrail
      Contact( #Stopper.ReleaseMemory )
      I_Contact( #Stopper.NextSensor )
      { S7_Templates := "time_type := Time" } #Stopper.ReachFaultTimer.TON(pt := #iReachFaultTimer, et =>)
      wire#w2
      Coil( #oReachFault )
      Coil( #io_Dev.ReachFault )
   END_RUNG
   RUNG wire#powerrail
      Contact( #oReachFault )
      I_Contact( #iSysInface.Reset )
   END_RUNG wire#w2
   // the same network as SCL:
   #Stopper.ReleaseFaultTimer.TON(IN := #Stopper.Valve AND #Stopper.Sensor, PT := #iReleaseFaultTimer);
   #oReleaseFault := #Stopper.ReleaseFaultTimer.Q OR (#oReleaseFault AND NOT #iSysInface.Reset);
   #io_Dev.ReleaseFault := #oReleaseFault;
   #Stopper.ReachFaultTimer.TON(IN := #Stopper.ReleaseMemory AND NOT #Stopper.NextSensor,
                           PT := #iReachFaultTimer);
   #oReachFault := #Stopper.ReachFaultTimer.Q OR (#oReachFault AND NOT #iSysInface.Reset);
   #io_Dev.ReachFault := #oReachFault;
END_REGION

REGION Network 9: 手动释放中 / Manual release
   RUNG wire#powerrail
      Contact( #iSysInface.ManualMode )
      Contact( #io_Dev.ReleasePB )
      I_Contact( #Stopper.ReleaseClear )
      I_Contact( #Stopper.Valve )
      Coil( #oNotClear )
      Coil( #io_Dev.NoClear )
   END_RUNG
   RUNG wire#powerrail
      Contact( #iSysInface.ManualMode )
      R_Coil( #io_Dev.AutoTrg )
   END_RUNG
   // the same network as SCL:
   #oNotClear := #iSysInface.ManualMode AND #io_Dev.ReleasePB AND NOT #Stopper.ReleaseClear AND NOT #Stopper.Valve;
   #io_Dev.NoClear := #oNotClear;
   IF #iSysInface.ManualMode THEN #io_Dev.AutoTrg := FALSE; END_IF;
END_REGION
END_FUNCTION_BLOCK

FUNCTION_BLOCK "FB_AteqF620"   // FB4080, SCL
TITLE = ATEQ F620 FB
{ S7_Optimized_Access := 'FALSE' }
AUTHOR : Chaoyao.Zheng
FAMILY : LeakTester
VERSION : 1.0
// stored: AutoNumber false, SetENOAutomatically false
   VAR_INPUT
      iHWID_Slot1 { ExternalAccessible := 'False'; ExternalVisible := 'False'; ExternalWritable := 'False'} : HW_IO;   // Input1
      iHWID_Slot2 { ExternalAccessible := 'False'; ExternalVisible := 'False'; ExternalWritable := 'False'} : HW_IO;   // Input2
      iHWID_Slot3 { ExternalAccessible := 'False'; ExternalVisible := 'False'; ExternalWritable := 'False'} : HW_IO;   // Input3
      iHWID_Slot4 { ExternalAccessible := 'False'; ExternalVisible := 'False'; ExternalWritable := 'False'} : HW_IO;   // Input4
      iHWID_Slot5 { ExternalAccessible := 'False'; ExternalVisible := 'False'; ExternalWritable := 'False'} : HW_IO;   // Output1
      iHWID_Slot6 { ExternalAccessible := 'False'; ExternalVisible := 'False'; ExternalWritable := 'False'} : HW_IO;   // Output2
      iHWID_Slot7 { ExternalAccessible := 'False'; ExternalVisible := 'False'; ExternalWritable := 'False'} : HW_IO;   // Output3
      iHWID_Slot8 { ExternalAccessible := 'False'; ExternalVisible := 'False'; ExternalWritable := 'False'} : HW_IO;   // Output4
      iSysRun { ExternalAccessible := 'False'; ExternalVisible := 'False'; ExternalWritable := 'False'} : Bool;
      iReset { ExternalAccessible := 'False'; ExternalVisible := 'False'; ExternalWritable := 'False'} : Bool;
      iAuto { ExternalAccessible := 'False'; ExternalVisible := 'False'; ExternalWritable := 'False'} : Bool;
      iManual { ExternalAccessible := 'False'; ExternalVisible := 'False'; ExternalWritable := 'False'} : Bool;
      iTimeout { ExternalAccessible := 'False'; ExternalVisible := 'False'; ExternalWritable := 'False'} : Time := T#5S;
   END_VAR
   VAR_OUTPUT
      oDeviceReady { ExternalAccessible := 'False'; ExternalVisible := 'False'; ExternalWritable := 'False'} : Bool;
      oReady { ExternalAccessible := 'False'; ExternalVisible := 'False'; ExternalWritable := 'False'} : Bool;
      oError { ExternalAccessible := 'False'; ExternalVisible := 'False'; ExternalWritable := 'False'} : Bool;
      oSetProgOk { ExternalAccessible := 'False'; ExternalVisible := 'False'; ExternalWritable := 'False'} : Bool;
      oMeasureOk { ExternalAccessible := 'False'; ExternalVisible := 'False'; ExternalWritable := 'False'} : Bool;
      oErrorCode { ExternalAccessible := 'False'; ExternalVisible := 'False'; ExternalWritable := 'False'} : UInt;
      oFillTime : Real;
      oStabTime : Real;
      oTeatTime : Real;
      oDumpTime : Real;
      oResult { ExternalAccessible := 'False'; ExternalVisible := 'False'; ExternalWritable := 'False'} : Struct
         PassPart : Bool;
         FailTestPart : Bool;
         FailRefPart : Bool;
         Alarm : Bool;
         PressureError : Bool;
         PartRecoverable : Bool;
         CalibError : Bool;
         CalibCheckError : Bool;
         AtrFault : Bool;
         Leak : Struct
            Value : Real;
            Unit : String[10];
         END_STRUCT;
      END_STRUCT;
      oPressure { ExternalAccessible := 'False'; ExternalVisible := 'False'; ExternalWritable := 'False'} : Struct
         Value : Real;
         Unit : String[10];
      END_STRUCT;
      oActProgStep { ExternalAccessible := 'False'; ExternalVisible := 'False'; ExternalWritable := 'False'} : UInt;
      oActProgNo { ExternalAccessible := 'False'; ExternalVisible := 'False'; ExternalWritable := 'False'} : UInt;
      oElapsedTime { ExternalAccessible := 'False'; ExternalVisible := 'False'; ExternalWritable := 'False'} : Time;
   END_VAR
   VAR_IN_OUT
      ioSetProg { ExternalAccessible := 'False'; ExternalVisible := 'False'; ExternalWritable := 'False'} : Bool;
      ioMeasure { ExternalAccessible := 'False'; ExternalVisible := 'False'; ExternalWritable := 'False'} : Bool;
      ioSpecialCycle : Bool;
      ioReadProTime : Bool;
   END_VAR
   VAR
      sHMI : "RCS_typeAteqF620Visual";
      sAuto { ExternalAccessible := 'False'; ExternalVisible := 'False'; ExternalWritable := 'False'} : Struct
         Set : Struct
            ProgNo : UInt;   // document name
         END_STRUCT;
      END_STRUCT;
      sHelp { ExternalAccessible := 'False'; ExternalVisible := 'False'; ExternalWritable := 'False'} : Struct
         First : Bool := FALSE;
         AutoOld : Bool;
         ManualOld : Bool;
         ResetRis : Bool;
         ResetOld : Bool;
         SetProgRis : Bool;
         SetProgOld : Bool;
         SetProgAct : Bool;
         MeasureRis : Bool;
         MeasureOld : Bool;
         MeasureAct : Bool;
         EnableTime : Bool;
         Abort : Bool;
         OrderCnt : UInt;
         "Step" : Array[1..2] of UInt;
         CmdTimer { S7_SetPoint := 'True'} : TON_TIME;
         Set : Struct
            ProgNo : UInt;   // document name
         END_STRUCT;
      END_STRUCT;
      sRecv { ExternalAccessible := 'False'; ExternalVisible := 'False'; ExternalWritable := 'False'} : Struct
         Echo : Struct
            Reset : Bool;
            Start : Bool;
            StartSpec : Bool;
            ProgramSel : Bool;
            ReadPara : Bool;
            ReadLastResult : Bool;
            Status : UInt;
         END_STRUCT;
         Result : Struct
            PassPart : Bool;
            FailTestPart : Bool;
            FailRefPart : Bool;
            Alarm : Bool;
            PressureError : Bool;
            PartRecoverable : Bool;
            CalibError : Bool;
            CalibCheckError : Bool;
            AtrFault : Bool;
            Leak : Struct
               Value : Real;
               Unit : String[10];
            END_STRUCT;
         END_STRUCT;
         CycleEnd : Bool;
         ErrorCode : UInt;
         ActProgram : UInt;
         ResultCnt : UInt;
         ActTestType : UInt;
         ActProgStep : UInt;
         ActPressure : UDInt;
         PressureUnitCode : UDInt;
         ActLeak : UDInt;
         LeakUnitCode : UDInt;
         FillTime : UDInt;
         StabTime : UDInt;
         TeatTime : UDInt;
         DumpTime : UDInt;
      END_STRUCT;
      sSend { ExternalAccessible := 'False'; ExternalVisible := 'False'; ExternalWritable := 'False'} : Struct
         Reset : Bool;
         Start : Bool;
         StartSpec : Bool;
         ProgramSel : Bool;
         ReadPara : Bool;
         ReadLastResult : Bool;
         ProgNo : UInt;
      END_STRUCT;
      sArrayInput { ExternalAccessible := 'False'; ExternalVisible := 'False'; ExternalWritable := 'False'} : Array[1..#cSlotAmount, 1..#cFieldbusBytes] of Byte;
      sArrayOutput { ExternalAccessible := 'False'; ExternalVisible := 'False'; ExternalWritable := 'False'} : Array[1..#cSlotAmount, 1..#cFieldbusBytes] of Byte;
      SpecialCycleStep : Int;
      ReadProTimeStep : Int;
      IEC_Timer_0_Instance { S7_SetPoint := 'True'} : TON_TIME;
      IEC_Timer_1_Instance { S7_SetPoint := 'True'} : TON_TIME;
      IEC_Timer_0_Instance_1 { S7_SetPoint := 'True'} : TON_TIME;
      IEC_Timer_1_Instance_1 { S7_SetPoint := 'True'} : TON_TIME;
      IEC_Timer_2_Instance_1 { S7_SetPoint := 'True'} : TON_TIME;
   END_VAR
   VAR_TEMP
      tIndex : UInt;
      tLoop : Int;
      tZero : Byte;
      tRetval : Struct
         LocallyErrID : Word;
         DPRD : Array[1..#cSlotAmount] of Int;
         DPWR : Array[1..#cSlotAmount] of Int;
         FILL : Int;
      END_STRUCT;
   END_VAR
   VAR CONSTANT
      cSlotAmount : UInt := 4;
      cFieldbusBytes : UInt := 64;
   END_VAR
BEGIN
   REGION Description header
       //================================================================================
       // (C) Ruhlamat Automation Technologies (Suzhou) Co.,Ltd.
       //--------------------------------------------------------------------------------
       // TargetSystem: ATEQ F620(COMX 100XX-PNS)
       // Engineering : TIA Portal V15 SP1
       // Author      : Chaoyao.Zheng
       //--------------------------------------------------------------------------------
       // Moduleversions:
       // V1.0 2020-08-24 - Chaoyao
       // - Initial version
       //================================================================================
   END_REGION
   REGION Error code explanation
       //  100: DPRD_DAT error occurred                                    
       //  101: DPWR_DAT error occurred                                    
       //  102: GET_ERR_ID error occurred                                  
       //  200: Order while FB not ready (oReady=FALSE)                    
       //  201: Several orders set at the same time                        
       //  202: Program number is not valid (1-128)                        
       //  203: Command error occurred                                     
       //  204: Command timeout                                            
   END_REGION

   (* FB Init *)
   IF NOT #sHelp.First THEN
       (* initialize outputs *)
       #sHelp.Abort := FALSE;
       #oDeviceReady := FALSE;
       #oReady := FALSE;
       #oSetProgOk := FALSE;
       #oMeasureOk := FALSE;
       #oErrorCode := 0;
       #oElapsedTime := T#0s;
       #tZero := 0;
       #tRetval.FILL := FILL(BVAL := #tZero, BLK => #oResult);
       #sHMI.Status.InstanceName := GetInstanceName(0);
       #sHelp.First := TRUE;
   ELSE
       (* reset fieldbus output *)
       FOR #tLoop := 1 TO UINT_TO_INT(#cSlotAmount) DO
           UFILL_BLK(IN := 0,
                     COUNT := #cFieldbusBytes,
                     OUT => #sArrayOutput[#tLoop, 01]);
       END_FOR;

       (* cyclic read tester input *)
       #tRetval.DPRD[1] := DPRD_DAT(LADDR := #iHWID_Slot1,
                                    RECORD => #sArrayInput[1]);
       #tRetval.DPRD[2] := DPRD_DAT(LADDR := #iHWID_Slot2,
                                    RECORD => #sArrayInput[2]);
       #tRetval.DPRD[3] := DPRD_DAT(LADDR := #iHWID_Slot3,
                                    RECORD => #sArrayInput[3]);
       #tRetval.DPRD[4] := DPRD_DAT(LADDR := #iHWID_Slot4,
                                    RECORD => #sArrayInput[4]);
       IF (#tRetval.DPRD[1] <> 0) OR (#tRetval.DPRD[2] <> 0) OR (#tRetval.DPRD[3] <> 0) OR (#tRetval.DPRD[4] <> 0) THEN
           #oErrorCode := 100; // Error cyclic read
       END_IF;

       (* move input bytes to static bits *)
       #sRecv.Echo.Reset := #sArrayInput[1, 01].%X0;
       #sRecv.Echo.Start := #sArrayInput[1, 01].%X1;
       #sRecv.Echo.StartSpec := #sArrayInput[1, 01].%X2;
       #sRecv.Echo.ProgramSel := #sArrayInput[1, 01].%X3;
       #sRecv.Echo.ReadPara := #sArrayInput[1, 02].%X5;
       #sRecv.Echo.ReadLastResult := #sArrayInput[1, 02].%X7;
       #sRecv.Result.PassPart := #sArrayInput[1, 13].%X0;
       #sRecv.Result.FailTestPart := #sArrayInput[1, 13].%X1;
       #sRecv.Result.FailRefPart := #sArrayInput[1, 13].%X2;
       #sRecv.Result.Alarm := #sArrayInput[1, 13].%X3;
       #sRecv.Result.PressureError := #sArrayInput[1, 13].%X4;
       #sRecv.CycleEnd := #sArrayInput[1, 13].%X5;
       #sRecv.Result.PartRecoverable := #sArrayInput[1, 13].%X6;
       #sRecv.Result.CalibError := #sArrayInput[1, 13].%X7;
       #sRecv.Result.CalibCheckError := #sArrayInput[1, 14].%X0;
       #sRecv.Result.AtrFault := #sArrayInput[1, 14].%X1;
       #sRecv.Result.Leak.Value := DINT_TO_REAL(#sRecv.ActLeak) / 1000.0;
       #oFillTime := DINT_TO_REAL(#sRecv.FillTime) / 1000.0;
       #oStabTime := DINT_TO_REAL(#sRecv.StabTime) / 1000.0;
       #oTeatTime := DINT_TO_REAL(#sRecv.TeatTime) / 1000.0;
       #oDumpTime := DINT_TO_REAL(#sRecv.DumpTime) / 1000.0;
       #sRecv.Echo.Status.%B0 := #sArrayInput[1, 01];
       #sRecv.Echo.Status.%B1 := #sArrayInput[1, 02];
       #sRecv.ErrorCode.%B0 := #sArrayInput[1, 03];
       #sRecv.ErrorCode.%B1 := #sArrayInput[1, 04];
       #sRecv.ActProgram.%B0 := #sArrayInput[1, 07];
       #sRecv.ActProgram.%B1 := #sArrayInput[1, 08];
       #sRecv.ActProgStep.%B0 := #sArrayInput[1, 15];
       #sRecv.ActProgStep.%B1 := #sArrayInput[1, 16];
       #sRecv.ActPressure.%B0 := #sArrayInput[1, 17];
       #sRecv.ActPressure.%B1 := #sArrayInput[1, 18];
       #sRecv.ActPressure.%B2 := #sArrayInput[1, 19];
       #sRecv.ActPressure.%B3 := #sArrayInput[1, 20];
       #sRecv.PressureUnitCode.%B0 := #sArrayInput[1, 21];
       #sRecv.PressureUnitCode.%B1 := #sArrayInput[1, 22];
       #sRecv.PressureUnitCode.%B2 := #sArrayInput[1, 23];
       #sRecv.PressureUnitCode.%B3 := #sArrayInput[1, 24];
       #sRecv.ActLeak.%B0 := #sArrayInput[1, 25];
       #sRecv.ActLeak.%B1 := #sArrayInput[1, 26];
       #sRecv.ActLeak.%B2 := #sArrayInput[1, 27];
       #sRecv.ActLeak.%B3 := #sArrayInput[1, 28];
       #sRecv.LeakUnitCode.%B0 := #sArrayInput[1, 29];
       #sRecv.LeakUnitCode.%B1 := #sArrayInput[1, 30];
       #sRecv.LeakUnitCode.%B2 := #sArrayInput[1, 31];
       #sRecv.LeakUnitCode.%B3 := #sArrayInput[1, 32];
       #sRecv.FillTime.%B0 := #sArrayInput[1, 35];
       #sRecv.FillTime.%B1 := #sArrayInput[1, 36];
       #sRecv.FillTime.%B2 := #sArrayInput[1, 37];
       #sRecv.FillTime.%B3 := #sArrayInput[1, 38];
       #sRecv.StabTime.%B0 := #sArrayInput[1, 41];
       #sRecv.StabTime.%B1 := #sArrayInput[1, 42];
       #sRecv.StabTime.%B2 := #sArrayInput[1, 43];
       #sRecv.StabTime.%B3 := #sArrayInput[1, 44];
       #sRecv.TeatTime.%B0 := #sArrayInput[1, 47];
       #sRecv.TeatTime.%B1 := #sArrayInput[1, 48];
       #sRecv.TeatTime.%B2 := #sArrayInput[1, 49];
       #sRecv.TeatTime.%B3 := #sArrayInput[1, 50];
       #sRecv.DumpTime.%B0 := #sArrayInput[1, 53];
       #sRecv.DumpTime.%B1 := #sArrayInput[1, 54];
       #sRecv.DumpTime.%B2 := #sArrayInput[1, 55];
       #sRecv.DumpTime.%B3 := #sArrayInput[1, 56];



       CASE #sRecv.LeakUnitCode OF
           0000:
               #sRecv.Result.Leak.Unit := 'cm3/s';
           1000:
               #sRecv.Result.Leak.Unit := 'cm3/min';
           2000:
               #sRecv.Result.Leak.Unit := 'cm3/h';
           3000:
               #sRecv.Result.Leak.Unit := 'mm3/h';
           4000:
               #sRecv.Result.Leak.Unit := 'Pa';
           5000:
               #sRecv.Result.Leak.Unit := 'Pa/s';
           6000:
               #sRecv.Result.Leak.Unit := 'Pa';
           7000:
               #sRecv.Result.Leak.Unit := 'Pa';
           8000:
               #sRecv.Result.Leak.Unit := 'Pa/s';
           9000:
               #sRecv.Result.Leak.Unit := 'Pa/s';
           11000:
               #sRecv.Result.Leak.Unit := 'bar';
           12000:
               #sRecv.Result.Leak.Unit := 'KPa';
           13000:
               #sRecv.Result.Leak.Unit := 'psi';
           14000:
               #sRecv.Result.Leak.Unit := 'mbar';
           15000:
               #sRecv.Result.Leak.Unit := 'MPa';
           43000:
               #sRecv.Result.Leak.Unit := 'Pa';
           44000:
               #sRecv.Result.Leak.Unit := 'Pa';
           45000:
               #sRecv.Result.Leak.Unit := 'Pa/s';
           46000:
               #sRecv.Result.Leak.Unit := 'In3/s';
           47000:
               #sRecv.Result.Leak.Unit := 'In3/min';
           48000:
               #sRecv.Result.Leak.Unit := 'In3/h';
           49000:
               #sRecv.Result.Leak.Unit := 'Ft3/h';
           50000:
               #sRecv.Result.Leak.Unit := 'mL/s';
           51000:
               #sRecv.Result.Leak.Unit := 'mL/min';
           52000:
               #sRecv.Result.Leak.Unit := 'mL/h';
           58000:
               #sRecv.Result.Leak.Unit := 'cm3/s';
           59000:
               #sRecv.Result.Leak.Unit := 'cm3/min';
           60000:
               #sRecv.Result.Leak.Unit := 'cm3/h';
           76000:
               #sRecv.Result.Leak.Unit := 'Ft3/s';
           77000:
               #sRecv.Result.Leak.Unit := 'Ft3/min';
           84000:
               #sRecv.Result.Leak.Unit := 'sccm';
           ELSE
               ;
       END_CASE;

       (* detection mode change *)
       IF NOT #iSysRun OR (#iManual XOR #sHelp.ManualOld) OR (#iAuto XOR #sHelp.AutoOld) THEN
           #sHMI.Trigger.SetProg := FALSE;
           #sHMI.Trigger.Measure := FALSE;
           #ioSetProg := FALSE;
           #ioMeasure := FALSE;
           (* reset outputs *)
           // Todo
       END_IF;
       #sHelp.ManualOld := #iManual;
       #sHelp.AutoOld := #iAuto;

       (* detection rising edges of inputs *)
       IF #iManual THEN
           #ioSetProg := FALSE;
           #ioMeasure := FALSE;
       ELSIF #iAuto THEN
           #sHMI.Trigger.SetProg := FALSE;
           #sHMI.Trigger.Measure := FALSE;
       END_IF;
       #sHelp.ResetRis := NOT #sHelp.ResetOld AND #iReset;
       #sHelp.ResetOld := #iReset;
       #sHelp.SetProgRis := NOT #sHelp.SetProgOld AND (#sHMI.Trigger.SetProg OR #ioSetProg);
       #sHelp.SetProgOld := #sHMI.Trigger.SetProg OR #ioSetProg;
       #sHelp.MeasureRis := NOT #sHelp.MeasureOld AND (#sHMI.Trigger.Measure OR #ioMeasure);
       #sHelp.MeasureOld := #sHMI.Trigger.Measure OR #ioMeasure;

       (* order handling *)
       #sHelp.OrderCnt := 0;
       IF #sHelp.SetProgOld THEN
           #sHelp.OrderCnt := #sHelp.OrderCnt + 1;
       END_IF;
       IF #sHelp.MeasureOld THEN
           #sHelp.OrderCnt := #sHelp.OrderCnt + 1;
       END_IF;
       IF (#sHelp.OrderCnt > 1) AND (#oErrorCode = 0) THEN
           #oErrorCode := 201; // twice command request
       END_IF;
       IF (#oErrorCode = 0) AND NOT #oReady THEN
           IF #sHelp.SetProgRis OR #sHelp.MeasureRis THEN
               #oErrorCode := 200; // command while not ready
           END_IF;
       END_IF;

       (* error clear *)
       IF (#sHelp.OrderCnt = 0) THEN
           IF #sHelp.ResetRis THEN
               #oErrorCode := 0;
               #sSend.Reset := TRUE;
           ELSE
               #sSend.Reset := FALSE;
           END_IF;
       END_IF;

       (* check timeout *)
       #sHelp.CmdTimer(IN := #sHelp.EnableTime,
                       PT := #iTimeout);
       (* Sequence --- SetProg *)
       REGION SetProg
           #tIndex := 1;

           IF (#oErrorCode = 0) AND #sHelp.SetProgRis THEN
               #tZero := 0;
               #tRetval.FILL := FILL(BVAL := #tZero, BLK => #oResult);
               IF #iAuto THEN
                   #sHelp.Set := #sAuto.Set;
               ELSE
                   #sHelp.Set := #sHMI.Set;
               END_IF;
               IF (#sHelp.Set.ProgNo >= 1) AND (#sHelp.Set.ProgNo <= 128) THEN
                   #sHelp.Abort := FALSE;
                   #sHelp.SetProgAct := TRUE;
                   #sHelp.Step[#tIndex] := 0;
               ELSE
                   #oErrorCode := 202;
               END_IF;
           END_IF;

           IF NOT #sHelp.SetProgOld THEN
               #oSetProgOk := FALSE;
               IF #sHelp.SetProgAct THEN
                   #sHelp.Abort := TRUE;
               END_IF;
           END_IF;

           IF #sHelp.SetProgAct THEN
               CASE #sHelp.Step[#tIndex] OF
                   0:  (* check error code *)
                       IF #sRecv.ErrorCode <> 16#0000 THEN
                           #sHelp.Step[#tIndex] := 1;
                       ELSE
                           #sHelp.Step[#tIndex] := 4;
                       END_IF;

                   1:  (* start order *)
                       IF #sRecv.Echo.Status = 16#0000 THEN
                           #sSend.Reset := TRUE;
                           #sHelp.EnableTime := FALSE;
                           #sHelp.Step[#tIndex] := #sHelp.Step[#tIndex] + 1;
                       END_IF;

                   2:  (* order accepted *)
                       IF #sRecv.Echo.Reset AND #sRecv.ErrorCode = 16#FFFF THEN
                           #sHelp.EnableTime := FALSE;
                           #sHelp.Step[#tIndex] := #sHelp.Step[#tIndex] + 1;
                       ELSE
                           #sHelp.EnableTime := TRUE;
                           IF #sHelp.CmdTimer.Q THEN
                               #oErrorCode := 204;
                               #sHelp.Step[#tIndex] := 99;
                           END_IF;
                       END_IF;

                   3:  (* order finished *)
                       IF #sRecv.Echo.Reset AND #sRecv.ErrorCode <> 16#FFFF THEN
                           #sSend.Reset := FALSE;
                           #sHelp.EnableTime := FALSE;
                           IF #sRecv.ErrorCode = 16#0000 THEN
                               #sHelp.Step[#tIndex] := #sHelp.Step[#tIndex] + 1;
                           ELSE
                               #oErrorCode := 203;
                               #sHelp.Step[#tIndex] := 99;
                           END_IF;
                       ELSE
                           #sHelp.EnableTime := TRUE;
                           IF #sHelp.CmdTimer.Q THEN
                               #oErrorCode := 204;
                               #sHelp.Step[#tIndex] := 99;
                           END_IF;
                       END_IF;

                   4:  (* start order *)
                       IF (#sRecv.Echo.Status = 16#0000) THEN
                           #sSend.ProgNo := #sHelp.Set.ProgNo - 1;
                           #sSend.ProgramSel := TRUE;
                           #sHelp.EnableTime := FALSE;
                           #sHelp.Step[#tIndex] := #sHelp.Step[#tIndex] + 1;
                       END_IF;

                   5:  (* order accepted *)
                       IF #sRecv.Echo.ProgramSel AND #sRecv.ErrorCode = 16#FFFF THEN
                           #sHelp.EnableTime := FALSE;
                           #sHelp.Step[#tIndex] := #sHelp.Step[#tIndex] + 1;
                       ELSE
                           #sHelp.EnableTime := TRUE;
                           IF #sHelp.CmdTimer.Q THEN
                               #oErrorCode := 204;
                               #sHelp.Step[#tIndex] := 995;
                           END_IF;
                       END_IF;

                   6:  (* order finished *)
                       IF #sRecv.Echo.ProgramSel AND #sRecv.ErrorCode <> 16#FFFF THEN
                           #sSend.ProgramSel := FALSE;
                           #sHelp.EnableTime := FALSE;
                           IF #sRecv.ErrorCode = 16#0000 THEN
                               #sHelp.Step[#tIndex] := 996;
                           ELSE
                               #oErrorCode := 203;
                               #sHelp.Step[#tIndex] := 997;
                           END_IF;
                       ELSE
                           #sHelp.EnableTime := TRUE;
                           IF #sHelp.CmdTimer.Q THEN
                               #oErrorCode := 204;
                               #sHelp.Step[#tIndex] := 998;
                           END_IF;
                       END_IF;

                   99,995,996,997,998,999:
                       #sSend.Reset := FALSE;
                       #sSend.ProgramSel := FALSE;
                       #sHelp.SetProgAct := FALSE;
                       #sHMI.Trigger.SetProg := FALSE;
                       #sHelp.Abort := FALSE;
                       IF #oErrorCode = 0 THEN
                           #oSetProgOk := TRUE;
                       END_IF;
               END_CASE;
           END_IF;
       END_REGION
       (* Sequence --- Measure *)
       REGION Measure
           #tIndex := 2;

           IF (#oErrorCode = 0) AND #sHelp.MeasureRis THEN
               #tZero := 0;
               #tRetval.FILL := FILL(BVAL := #tZero, BLK => #oResult);
               IF #iAuto THEN
                   #sHelp.Set := #sAuto.Set;
               ELSE
                   #sHelp.Set := #sHMI.Set;
               END_IF;
               #sHelp.Abort := FALSE;
               #sHelp.MeasureAct := TRUE;
               #sHelp.Step[#tIndex] := 0;
           END_IF;

           IF NOT #sHelp.MeasureOld THEN
               #oMeasureOk := FALSE;
               IF #sHelp.MeasureAct THEN
                   #sHelp.Abort := TRUE;
               END_IF;
           END_IF;

           IF #sHelp.MeasureAct THEN
               CASE #sHelp.Step[#tIndex] OF
                   0:  (* check error code *)
                       IF #sRecv.ErrorCode <> 16#0000 THEN
                           #sHelp.Step[#tIndex] := 1;
                       ELSE
                           #sHelp.Step[#tIndex] := 4;
                       END_IF;

                   1:  (* start order *)
                       IF #sRecv.Echo.Status = 16#0000 THEN
                           #sSend.Reset := TRUE;
                           #sHelp.EnableTime := FALSE;
                           #sHelp.Step[#tIndex] := #sHelp.Step[#tIndex] + 1;
                       END_IF;

                   2:  (* order accepted *)
                       IF #sRecv.Echo.Reset AND #sRecv.ErrorCode = 16#FFFF THEN
                           #sHelp.EnableTime := FALSE;
                           #sHelp.Step[#tIndex] := #sHelp.Step[#tIndex] + 1;
                       ELSE
                           #sHelp.EnableTime := TRUE;
                           IF #sHelp.CmdTimer.Q THEN
                               #oErrorCode := 204;
                               #sHelp.Step[#tIndex] := 299;
                           END_IF;
                       END_IF;

                   3:  (* order finished *)
                       IF #sRecv.Echo.Reset AND #sRecv.ErrorCode <> 16#FFFF THEN
                           #sSend.Reset := FALSE;
                           #sHelp.EnableTime := FALSE;
                           IF #sRecv.ErrorCode = 16#0000 THEN
                               #sHelp.Step[#tIndex] := #sHelp.Step[#tIndex] + 1;
                           ELSE
                               #oErrorCode := 203;
                               #sHelp.Step[#tIndex] := 398;
                           END_IF;
                       ELSE
                           #sHelp.EnableTime := TRUE;
                           IF #sHelp.CmdTimer.Q THEN
                               #oErrorCode := 204;
                               #sHelp.Step[#tIndex] := 399;
                           END_IF;
                       END_IF;

                   4:  (* start order *)
                       IF (#sRecv.Echo.Status = 16#0000) THEN
                           #sSend.Start := TRUE;
                           #sHelp.EnableTime := FALSE;
                           #sHelp.Step[#tIndex] := #sHelp.Step[#tIndex] + 1;
                       END_IF;

                   5:  (* order accepted *)
                       IF #sRecv.Echo.Start AND #sRecv.ErrorCode = 16#FFFF THEN
                           #sHelp.EnableTime := FALSE;
                           #sHelp.Step[#tIndex] := #sHelp.Step[#tIndex] + 1;
                       ELSE
                           #sHelp.EnableTime := TRUE;
                           IF #sHelp.CmdTimer.Q THEN
                               #oErrorCode := 204;
                               #sHelp.Step[#tIndex] := 599;
                           END_IF;
                       END_IF;

